LIN {X 0,Y 474.62,Z 424.367,A -85,B 0,C 180,E1 -7430.451,E2 -7430.451} C_VEL
LIN {X 0,Y 474.556,Z 424.367,A -85,B 0,C 180,E1 -7433.225,E2 -7433.225} C_VEL
LIN {X 0,Y 473.902,Z 424.453,A -85,B 0,C 180,E1 -7433.934,E2 -7433.934} C_VEL
LIN {X 0,Y 471.059,Z 424.804,A -85,B 0,C 180,E1 -7435.086,E2 -7435.086} C_VEL
LIN {X 0,Y 468.658,Z 425.105,A -85,B 0,C 180,E1 -7436.015,E2 -7436.015} C_VEL
LIN {X 0,Y 467.644,Z 425.233,A -85,B 0,C 180,E1 -7436.732,E2 -7436.732} C_VEL
LIN {X 0,Y 467.57,Z 425.237,A -85,B 0,C 180,E1 -7436.975,E2 -7436.975} C_VEL
LIN {X 0,Y 467.568,Z 425.238,A -85,B 0,C 180,E1 -7439.266,E2 -7439.266} C_VEL
LIN {X 0,Y 467.577,Z 425.245,A -85,B 0,C 180,E1 -7442.475,E2 -7442.475} C_VEL
LIN {X 0,Y 467.57,Z 425.238,A -85,B 0,C 180,E1 -7445.11,E2 -7445.11} C_VEL
LIN {X 0,Y 467.536,Z 425.244,A -85,B 0,C 180,E1 -7447.926,E2 -7447.926} C_VEL
LIN {X 0,Y 467.622,Z 425.236,A -85,B 0,C 180,E1 -7450.692,E2 -7450.692} C_VEL
LIN {X 0,Y 467.639,Z 425.235,A -85,B 0,C 180,E1 -7454.305,E2 -7454.305} C_VEL
LIN {X 0,Y 467.658,Z 425.228,A -85,B 0,C 180,E1 -7457.854,E2 -7457.854} C_VEL
LIN {X 0,Y 467.669,Z 425.225,A -85,B 0,C 180,E1 -7461.357,E2 -7461.357} C_VEL
LIN {X 0,Y 467.714,Z 425.222,A -85,B 0,C 180,E1 -7463.962,E2 -7463.962} C_VEL
LIN {X 0,Y 467.852,Z 425.202,A -85,B 0,C 180,E1 -7467.417,E2 -7467.417} C_VEL
LIN {X 0,Y 467.88,Z 425.201,A -85,B 0,C 180,E1 -7470,E2 -7470} C_VEL
LIN {X 0,Y 467.848,Z 425.21,A -85,B 0,C 180,E1 -7472.583,E2 -7472.583} C_VEL
LIN {X 0,Y 467.741,Z 425.219,A -85,B 0,C 180,E1 -7476.037,E2 -7476.037} C_VEL
LIN {X 0,Y 467.669,Z 425.232,A -85,B 0,C 180,E1 -7478.643,E2 -7478.643} C_VEL
LIN {X 0,Y 467.657,Z 425.23,A -85,B 0,C 180,E1 -7482.145,E2 -7482.145} C_VEL
LIN {X 0,Y 467.64,Z 425.229,A -85,B 0,C 180,E1 -7485.695,E2 -7485.695} C_VEL
LIN {X 0,Y 467.623,Z 425.231,A -85,B 0,C 180,E1 -7489.307,E2 -7489.307} C_VEL
LIN {X 0,Y 467.535,Z 425.244,A -85,B 0,C 180,E1 -7492.074,E2 -7492.074} C_VEL
LIN {X 0,Y 467.583,Z 425.24,A -85,B 0,C 180,E1 -7494.888,E2 -7494.888} C_VEL
LIN {X 0,Y 467.58,Z 425.237,A -85,B 0,C 180,E1 -7497.771,E2 -7497.771} C_VEL
LIN {X 0,Y 467.568,Z 425.24,A -85,B 0,C 180,E1 -7501.045,E2 -7501.045} C_VEL
LIN {X 0,Y 467.588,Z 425.239,A -85,B 0,C 180,E1 -7504.242,E2 -7504.242} C_VEL
LIN {X 0,Y 467.543,Z 425.242,A -85,B 0,C 180,E1 -7507.185,E2 -7507.185} C_VEL
LIN {X 0,Y 467.569,Z 425.242,A -85,B 0,C 180,E1 -7510.265,E2 -7510.265} C_VEL
LIN {X 0,Y 467.559,Z 425.248,A -85,B 0,C 180,E1 -7512.563,E2 -7512.563} C_VEL
LIN {X 0,Y 467.564,Z 425.241,A -85,B 0,C 180,E1 -7515.052,E2 -7515.052} C_VEL
LIN {X 0,Y 467.572,Z 425.246,A -85,B 0,C 180,E1 -7518.597,E2 -7518.597} C_VEL
LIN {X 0,Y 467.558,Z 425.239,A -85,B 0,C 180,E1 -7521.409,E2 -7521.409} C_VEL
LIN {X 0,Y 467.557,Z 425.243,A -85,B 0,C 180,E1 -7524.261,E2 -7524.261} C_VEL
LIN {X 0,Y 467.581,Z 425.237,A -85,B 0,C 180,E1 -7527.321,E2 -7527.321} C_VEL
LIN {X 0,Y 467.568,Z 425.245,A -85,B 0,C 180,E1 -7530.668,E2 -7530.668} C_VEL
LIN {X 0,Y 467.587,Z 425.237,A -85,B 0,C 180,E1 -7533.198,E2 -7533.198} C_VEL
LIN {X 0,Y 467.59,Z 425.242,A -85,B 0,C 180,E1 -7536.469,E2 -7536.469} C_VEL
LIN {X 0,Y 467.622,Z 425.231,A -85,B 0,C 180,E1 -7539.777,E2 -7539.777} C_VEL
LIN {X 0,Y 467.597,Z 425.241,A -85,B 0,C 180,E1 -7542.506,E2 -7542.506} C_VEL
LIN {X 0,Y 467.604,Z 425.235,A -85,B 0,C 180,E1 -7545.196,E2 -7545.196} C_VEL
LIN {X 0,Y 467.656,Z 425.227,A -85,B 0,C 180,E1 -7547.855,E2 -7547.855} C_VEL
LIN {X 0,Y 467.68,Z 425.224,A -85,B 0,C 180,E1 -7551.357,E2 -7551.357} C_VEL
LIN {X 0,Y 467.723,Z 425.219,A -85,B 0,C 180,E1 -7553.962,E2 -7553.962} C_VEL
LIN {X 0,Y 467.858,Z 425.202,A -85,B 0,C 180,E1 -7557.417,E2 -7557.417} C_VEL
LIN {X 0,Y 467.882,Z 425.2,A -85,B 0,C 180,E1 -7560,E2 -7560} C_VEL
LIN {X 0,Y 467.858,Z 425.209,A -85,B 0,C 180,E1 -7562.583,E2 -7562.583} C_VEL
LIN {X 0,Y 467.742,Z 425.217,A -85,B 0,C 180,E1 -7566.037,E2 -7566.037} C_VEL
LIN {X 0,Y 467.68,Z 425.232,A -85,B 0,C 180,E1 -7568.643,E2 -7568.643} C_VEL
LIN {X 0,Y 467.656,Z 425.229,A -85,B 0,C 180,E1 -7572.146,E2 -7572.146} C_VEL
LIN {X 0,Y 467.639,Z 425.229,A -85,B 0,C 180,E1 -7575.695,E2 -7575.695} C_VEL
LIN {X 0,Y 467.613,Z 425.24,A -85,B 0,C 180,E1 -7578.763,E2 -7578.763} C_VEL
LIN {X 0,Y 467.58,Z 425.238,A -85,B 0,C 180,E1 -7581.268,E2 -7581.268} C_VEL
LIN {X 0,Y 467.568,Z 425.238,A -85,B 0,C 180,E1 -7583.944,E2 -7583.944} C_VEL
LIN {X 0,Y 467.59,Z 425.242,A -85,B 0,C 180,E1 -7586.802,E2 -7586.802} C_VEL
LIN {X 0,Y 467.553,Z 425.24,A -85,B 0,C 180,E1 -7589.738,E2 -7589.738} C_VEL
LIN {X 0,Y 467.583,Z 425.244,A -85,B 0,C 180,E1 -7592.759,E2 -7592.759} C_VEL
LIN {X 0,Y 467.553,Z 425.24,A -85,B 0,C 180,E1 -7595.89,E2 -7595.89} C_VEL
LIN {X 0,Y 467.576,Z 425.24,A -85,B 0,C 180,E1 -7599.146,E2 -7599.146} C_VEL
LIN {X 0,Y 467.587,Z 425.242,A -85,B 0,C 180,E1 -7602.567,E2 -7602.567} C_VEL
LIN {X 0,Y 467.571,Z 425.241,A -85,B 0,C 180,E1 -7605.053,E2 -7605.053} C_VEL
LIN {X 0,Y 467.589,Z 425.236,A -85,B 0,C 180,E1 -7607.44,E2 -7607.44} C_VEL
LIN {X 0,Y 467.582,Z 425.243,A -85,B 0,C 180,E1 -7610.856,E2 -7610.856} C_VEL
LIN {X 0,Y 467.558,Z 425.241,A -85,B 0,C 180,E1 -7614.262,E2 -7614.262} C_VEL
LIN {X 0,Y 467.583,Z 425.238,A -85,B 0,C 180,E1 -7617.321,E2 -7617.321} C_VEL
LIN {X 0,Y 467.57,Z 425.244,A -85,B 0,C 180,E1 -7620.668,E2 -7620.668} C_VEL
LIN {X 0,Y 467.64,Z 425.277,A -85,B 0,C 180,E1 -7621.958,E2 -7621.958} C_VEL
LIN {X 0,Y 470.44,Z 438.906,A -85,B 0,C 180,E1 -7624.327,E2 -7624.327} C_VEL
LIN {X 0,Y 470.495,Z 444.774,A -85,B 0,C 180,E1 -7625.276,E2 -7625.276} C_VEL
LIN {X 0,Y 469.437,Z 466.708,A -85,B 0,C 180,E1 -7628.726,E2 -7628.726} C_VEL
LIN {X 0,Y 468.659,Z 486.966,A -85,B 0,C 180,E1 -7631.871,E2 -7631.871} C_VEL
LIN {X 0,Y 468.408,Z 494.383,A -85,B 0,C 180,E1 -7633.004,E2 -7633.004} C_VEL
LIN {X 0,Y 471.057,Z 514.85,A -85,B 0,C 180,E1 -7633.441,E2 -7633.441} C_VEL
LIN {X 0,Y 470.187,Z 603.81,A -85,B 0,C 180,E1 -7634.92,E2 -7634.92} C_VEL
LIN {X 0,Y 469.824,Z 616.734,A -85,B 0,C 180,E1 -7635.296,E2 -7635.296} C_VEL
LIN {X 0,Y 469.33,Z 629.907,A -85,B 0,C 180,E1 -7635.861,E2 -7635.861} C_VEL
LIN {X 0,Y 468.901,Z 641.86,A -85,B 0,C 180,E1 -7636.567,E2 -7636.567} C_VEL
LIN {X 0,Y 468.404,Z 653.827,A -85,B 0,C 180,E1 -7637.474,E2 -7637.474} C_VEL
LIN {X 0,Y 467.977,Z 663.748,A -85,B 0,C 180,E1 -7638.413,E2 -7638.413} C_VEL
LIN {X 0,Y 467.505,Z 673.902,A -85,B 0,C 180,E1 -7639.607,E2 -7639.607} C_VEL
LIN {X 0,Y 467.18,Z 682.846,A -85,B 0,C 180,E1 -7640.912,E2 -7640.912} C_VEL
LIN {X 0,Y 466.959,Z 689.988,A -85,B 0,C 180,E1 -7642.215,E2 -7642.215} C_VEL
LIN {X 0,Y 466.803,Z 695.821,A -85,B 0,C 180,E1 -7643.552,E2 -7643.552} C_VEL
LIN {X 0,Y 466.779,Z 700.165,A -85,B 0,C 180,E1 -7644.817,E2 -7644.817} C_VEL
LIN {X 0,Y 466.701,Z 702.517,A -85,B 0,C 180,E1 -7645.682,E2 -7645.682} C_VEL
LIN {X 0,Y 466.758,Z 704.438,A -85,B 0,C 180,E1 -7646.547,E2 -7646.547} C_VEL
LIN {X 0,Y 466.775,Z 705.879,A -85,B 0,C 180,E1 -7647.411,E2 -7647.411} C_VEL
LIN {X 0,Y 466.698,Z 706.884,A -85,B 0,C 180,E1 -7648.274,E2 -7648.274} C_VEL
LIN {X 0,Y 466.633,Z 707.487,A -85,B 0,C 180,E1 -7649.137,E2 -7649.137} C_VEL
LIN {X 0,Y 466.624,Z 707.689,A -85,B 0,C 180,E1 -7650,E2 -7650} C_VEL
LIN {X 0,Y 466.634,Z 707.441,A -85,B 0,C 180,E1 -7650.863,E2 -7650.863} C_VEL
LIN {X 0,Y 466.699,Z 706.788,A -85,B 0,C 180,E1 -7651.726,E2 -7651.726} C_VEL
LIN {X 0,Y 466.792,Z 705.732,A -85,B 0,C 180,E1 -7652.589,E2 -7652.589} C_VEL
LIN {X 0,Y 466.772,Z 704.246,A -85,B 0,C 180,E1 -7653.453,E2 -7653.453} C_VEL
LIN {X 0,Y 466.712,Z 701.144,A -85,B 0,C 180,E1 -7654.751,E2 -7654.751} C_VEL
LIN {X 0,Y 466.783,Z 696.966,A -85,B 0,C 180,E1 -7656.05,E2 -7656.05} C_VEL
LIN {X 0,Y 466.939,Z 691.594,A -85,B 0,C 180,E1 -7657.351,E2 -7657.351} C_VEL
LIN {X 0,Y 467.099,Z 684.831,A -85,B 0,C 180,E1 -7658.654,E2 -7658.654} C_VEL
LIN {X 0,Y 467.348,Z 676.43,A -85,B 0,C 180,E1 -7659.959,E2 -7659.959} C_VEL
LIN {X 0,Y 467.714,Z 667.861,A -85,B 0,C 180,E1 -7661.046,E2 -7661.046} C_VEL
LIN {X 0,Y 468.107,Z 658.514,A -85,B 0,C 180,E1 -7662.024,E2 -7662.024} C_VEL
LIN {X 0,Y 468.56,Z 646.916,A -85,B 0,C 180,E1 -7663.002,E2 -7663.002} C_VEL
LIN {X 0,Y 469.023,Z 635.597,A -85,B 0,C 180,E1 -7663.762,E2 -7663.762} C_VEL
LIN {X 0,Y 469.521,Z 623.009,A -85,B 0,C 180,E1 -7664.41,E2 -7664.41} C_VEL
LIN {X 0,Y 469.953,Z 609.708,A -85,B 0,C 180,E1 -7664.894,E2 -7664.894} C_VEL
LIN {X 0,Y 470.286,Z 597.064,A -85,B 0,C 180,E1 -7665.188,E2 -7665.188} C_VEL
LIN {X 0,Y 471.024,Z 514.08,A -85,B 0,C 180,E1 -7666.577,E2 -7666.577} C_VEL
LIN {X 0,Y 468.283,Z 492.11,A -85,B 0,C 180,E1 -7667.095,E2 -7667.095} C_VEL
LIN {X 0,Y 469.001,Z 470.807,A -85,B 0,C 180,E1 -7670.39,E2 -7670.39} C_VEL
LIN {X 0,Y 469.616,Z 456.296,A -85,B 0,C 180,E1 -7672.666,E2 -7672.666} C_VEL
LIN {X 0,Y 470.349,Z 440.454,A -85,B 0,C 180,E1 -7675.205,E2 -7675.205} C_VEL
LIN {X 0,Y 469.688,Z 435.05,A -85,B 0,C 180,E1 -7676.131,E2 -7676.131} C_VEL
LIN {X 0,Y 467.625,Z 425.238,A -85,B 0,C 180,E1 -7677.952,E2 -7677.952} C_VEL
LIN {X 0,Y 467.572,Z 425.248,A -85,B 0,C 180,E1 -7681.045,E2 -7681.045} C_VEL
LIN {X 0,Y 467.592,Z 425.243,A -85,B 0,C 180,E1 -7684.242,E2 -7684.242} C_VEL
LIN {X 0,Y 467.552,Z 425.247,A -85,B 0,C 180,E1 -7687.186,E2 -7687.186} C_VEL
LIN {X 0,Y 467.581,Z 425.241,A -85,B 0,C 180,E1 -7690.265,E2 -7690.265} C_VEL
LIN {X 0,Y 467.59,Z 425.241,A -85,B 0,C 180,E1 -7692.567,E2 -7692.567} C_VEL
LIN {X 0,Y 467.569,Z 425.242,A -85,B 0,C 180,E1 -7695.053,E2 -7695.053} C_VEL
LIN {X 0,Y 467.577,Z 425.245,A -85,B 0,C 180,E1 -7698.597,E2 -7698.597} C_VEL
LIN {X 0,Y 467.562,Z 425.24,A -85,B 0,C 180,E1 -7701.41,E2 -7701.41} C_VEL
LIN {X 0,Y 467.561,Z 425.244,A -85,B 0,C 180,E1 -7704.262,E2 -7704.262} C_VEL
LIN {X 0,Y 467.585,Z 425.236,A -85,B 0,C 180,E1 -7707.321,E2 -7707.321} C_VEL
LIN {X 0,Y 467.554,Z 425.245,A -85,B 0,C 180,E1 -7710.672,E2 -7710.672} C_VEL
LIN {X 0,Y 467.538,Z 425.244,A -85,B 0,C 180,E1 -7713.195,E2 -7713.195} C_VEL
LIN {X 0,Y 467.559,Z 425.245,A -85,B 0,C 180,E1 -7716.056,E2 -7716.056} C_VEL
LIN {X 0,Y 467.551,Z 425.243,A -85,B 0,C 180,E1 -7718.853,E2 -7718.853} C_VEL
LIN {X 0,Y 467.595,Z 425.238,A -85,B 0,C 180,E1 -7721.601,E2 -7721.601} C_VEL
LIN {X 0,Y 467.58,Z 425.243,A -85,B 0,C 180,E1 -7724.303,E2 -7724.303} C_VEL
LIN {X 0,Y 467.644,Z 425.237,A -85,B 0,C 180,E1 -7727.854,E2 -7727.854} C_VEL
LIN {X 0,Y 467.632,Z 425.236,A -85,B 0,C 180,E1 -7731.356,E2 -7731.356} C_VEL
LIN {X 0,Y 467.696,Z 425.231,A -85,B 0,C 180,E1 -7733.962,E2 -7733.962} C_VEL
LIN {X 0,Y 467.669,Z 425.384,A -85,B 0,C 180,E1 -7736.877,E2 -7736.877} C_VEL
LIN {X 0,Y 468.59,Z 429.689,A -85,B 0,C 180,E1 -7738.039,E2 -7738.039} C_VEL
LIN {X 0,Y 471.558,Z 440.896,A -85,B 0,C 180,E1 -7738.372,E2 -7738.372} C_VEL
LIN {X 0,Y 470.383,Z 535.807,A -85,B 0,C 180,E1 -7740,E2 -7740} C_VEL
LIN {X 0,Y 470.125,Z 549.678,A -85,B 0,C 180,E1 -7740.428,E2 -7740.428} C_VEL
LIN {X 0,Y 469.901,Z 561.461,A -85,B 0,C 180,E1 -7740.964,E2 -7740.964} C_VEL
LIN {X 0,Y 469.503,Z 573.791,A -85,B 0,C 180,E1 -7741.716,E2 -7741.716} C_VEL
LIN {X 0,Y 468.962,Z 584.879,A -85,B 0,C 180,E1 -7742.577,E2 -7742.577} C_VEL
LIN {X 0,Y 468.572,Z 593.83,A -85,B 0,C 180,E1 -7743.439,E2 -7743.439} C_VEL
LIN {X 0,Y 468.172,Z 603.023,A -85,B 0,C 180,E1 -7744.52,E2 -7744.52} C_VEL
LIN {X 0,Y 467.851,Z 610.583,A -85,B 0,C 180,E1 -7745.603,E2 -7745.603} C_VEL
LIN {X 0,Y 467.55,Z 617.992,A -85,B 0,C 180,E1 -7746.907,E2 -7746.907} C_VEL
LIN {X 0,Y 467.272,Z 623.956,A -85,B 0,C 180,E1 -7748.215,E2 -7748.215} C_VEL
LIN {X 0,Y 467.067,Z 628.662,A -85,B 0,C 180,E1 -7749.527,E2 -7749.527} C_VEL
LIN {X 0,Y 466.951,Z 632.231,A -85,B 0,C 180,E1 -7750.844,E2 -7750.844} C_VEL
LIN {X 0,Y 466.833,Z 634.764,A -85,B 0,C 180,E1 -7752.167,E2 -7752.167} C_VEL
LIN {X 0,Y 466.732,Z 635.921,A -85,B 0,C 180,E1 -7753.054,E2 -7753.054} C_VEL
LIN {X 0,Y 466.701,Z 636.61,A -85,B 0,C 180,E1 -7753.942,E2 -7753.942} C_VEL
LIN {X 0,Y 466.716,Z 636.823,A -85,B 0,C 180,E1 -7755.475,E2 -7755.475} C_VEL
LIN {X 0,Y 466.695,Z 636.156,A -85,B 0,C 180,E1 -7756.626,E2 -7756.626} C_VEL
LIN {X 0,Y 466.725,Z 635.119,A -85,B 0,C 180,E1 -7757.527,E2 -7757.527} C_VEL
LIN {X 0,Y 466.83,Z 633.563,A -85,B 0,C 180,E1 -7758.476,E2 -7758.476} C_VEL
LIN {X 0,Y 466.92,Z 630.508,A -85,B 0,C 180,E1 -7759.796,E2 -7759.796} C_VEL
LIN {X 0,Y 467.078,Z 626.161,A -85,B 0,C 180,E1 -7761.169,E2 -7761.169} C_VEL
LIN {X 0,Y 467.305,Z 620.456,A -85,B 0,C 180,E1 -7762.551,E2 -7762.551} C_VEL
LIN {X 0,Y 467.609,Z 613.177,A -85,B 0,C 180,E1 -7763.941,E2 -7763.941} C_VEL
LIN {X 0,Y 467.967,Z 605.626,A -85,B 0,C 180,E1 -7765.104,E2 -7765.104} C_VEL
LIN {X 0,Y 468.37,Z 596.274,A -85,B 0,C 180,E1 -7766.273,E2 -7766.273} C_VEL
LIN {X 0,Y 468.81,Z 585.82,A -85,B 0,C 180,E1 -7767.329,E2 -7767.329} C_VEL
LIN {X 0,Y 469.261,Z 575.69,A -85,B 0,C 180,E1 -7768.155,E2 -7768.155} C_VEL
LIN {X 0,Y 469.663,Z 563.942,A -85,B 0,C 180,E1 -7768.916,E2 -7768.916} C_VEL
LIN {X 0,Y 470.051,Z 550.522,A -85,B 0,C 180,E1 -7769.564,E2 -7769.564} C_VEL
LIN {X 0,Y 470.317,Z 538.201,A -85,B 0,C 180,E1 -7769.982,E2 -7769.982} C_VEL
LIN {X 0,Y 470.461,Z 522.713,A -85,B 0,C 180,E1 -7770.292,E2 -7770.292} C_VEL
LIN {X 0,Y 471.2,Z 439.643,A -85,B 0,C 180,E1 -7771.663,E2 -7771.663} C_VEL
LIN {X 0,Y 468.607,Z 429.284,A -85,B 0,C 180,E1 -7771.935,E2 -7771.935} C_VEL
LIN {X 0,Y 467.973,Z 427.129,A -85,B 0,C 180,E1 -7772.018,E2 -7772.018} C_VEL
LIN {X 0,Y 467.621,Z 425.239,A -85,B 0,C 180,E1 -7772.538,E2 -7772.538} C_VEL
LIN {X 0,Y 467.55,Z 425.244,A -85,B 0,C 180,E1 -7775.89,E2 -7775.89} C_VEL
LIN {X 0,Y 467.546,Z 425.241,A -85,B 0,C 180,E1 -7779.148,E2 -7779.148} C_VEL
LIN {X 0,Y 467.567,Z 425.238,A -85,B 0,C 180,E1 -7781.404,E2 -7781.404} C_VEL
LIN {X 0,Y 467.568,Z 425.239,A -85,B 0,C 180,E1 -7785.052,E2 -7785.052} C_VEL
LIN {X 0,Y 467.564,Z 425.242,A -85,B 0,C 180,E1 -7788.725,E2 -7788.725} C_VEL
LIN {X 0,Y 467.543,Z 425.243,A -85,B 0,C 180,E1 -7791.953,E2 -7791.953} C_VEL
LIN {X 0,Y 467.56,Z 425.239,A -85,B 0,C 180,E1 -7795.166,E2 -7795.166} C_VEL
LIN {X 0,Y 467.57,Z 425.237,A -85,B 0,C 180,E1 -7796.975,E2 -7796.975} C_VEL
LIN {X 0,Y 466.933,Z 425.318,A -85,B 0,C 180,E1 -7797.693,E2 -7797.693} C_VEL
LIN {X 0,Y 464.106,Z 425.677,A -85,B 0,C 180,E1 -7798.86,E2 -7798.86} C_VEL
LIN {X 0,Y 461.684,Z 425.981,A -85,B 0,C 180,E1 -7799.8,E2 -7799.8} C_VEL
LIN {X 0,Y 460.62,Z 426.11,A -85,B 0,C 180,E1 -7800.527,E2 -7800.527} C_VEL
LIN {X 0,Y 460.522,Z 426.119,A -85,B 0,C 180,E1 -7800.773,E2 -7800.773} C_VEL
LIN {X 0,Y 460.521,Z 426.116,A -85,B 0,C 180,E1 -7803.732,E2 -7803.732} C_VEL
LIN {X 0,Y 460.546,Z 426.118,A -85,B 0,C 180,E1 -7806.624,E2 -7806.624} C_VEL
LIN {X 0,Y 460.552,Z 426.112,A -85,B 0,C 180,E1 -7809.452,E2 -7809.452} C_VEL
LIN {X 0,Y 460.543,Z 426.118,A -85,B 0,C 180,E1 -7812.229,E2 -7812.229} C_VEL
LIN {X 0,Y 460.562,Z 426.113,A -85,B 0,C 180,E1 -7814.964,E2 -7814.964} C_VEL
LIN {X 0,Y 460.611,Z 426.112,A -85,B 0,C 180,E1 -7818.559,E2 -7818.559} C_VEL
LIN {X 0,Y 460.619,Z 426.104,A -85,B 0,C 180,E1 -7821.223,E2 -7821.223} C_VEL
LIN {X 0,Y 460.679,Z 426.097,A -85,B 0,C 180,E1 -7823.869,E2 -7823.869} C_VEL
LIN {X 0,Y 460.792,Z 426.082,A -85,B 0,C 180,E1 -7827.377,E2 -7827.377} C_VEL
LIN {X 0,Y 460.85,Z 426.077,A -85,B 0,C 180,E1 -7830,E2 -7830} C_VEL
LIN {X 0,Y 460.789,Z 426.089,A -85,B 0,C 180,E1 -7832.622,E2 -7832.622} C_VEL
LIN {X 0,Y 460.706,Z 426.096,A -85,B 0,C 180,E1 -7836.13,E2 -7836.13} C_VEL
LIN {X 0,Y 460.619,Z 426.108,A -85,B 0,C 180,E1 -7838.776,E2 -7838.776} C_VEL
LIN {X 0,Y 460.615,Z 426.112,A -85,B 0,C 180,E1 -7842.445,E2 -7842.445} C_VEL
LIN {X 0,Y 460.601,Z 426.108,A -85,B 0,C 180,E1 -7845.997,E2 -7845.997} C_VEL
LIN {X 0,Y 460.569,Z 426.11,A -85,B 0,C 180,E1 -7849.615,E2 -7849.615} C_VEL
LIN {X 0,Y 460.511,Z 426.124,A -85,B 0,C 180,E1 -7852.428,E2 -7852.428} C_VEL
LIN {X 0,Y 460.549,Z 426.113,A -85,B 0,C 180,E1 -7855.797,E2 -7855.797} C_VEL
LIN {X 0,Y 460.527,Z 426.119,A -85,B 0,C 180,E1 -7858.234,E2 -7858.234} C_VEL
LIN {X 0,Y 460.521,Z 426.116,A -85,B 0,C 180,E1 -7861.283,E2 -7861.283} C_VEL
LIN {X 0,Y 460.531,Z 426.122,A -85,B 0,C 180,E1 -7864.505,E2 -7864.505} C_VEL
LIN {X 0,Y 460.498,Z 426.118,A -85,B 0,C 180,E1 -7867.623,E2 -7867.623} C_VEL
LIN {X 0,Y 460.526,Z 426.118,A -85,B 0,C 180,E1 -7871.011,E2 -7871.011} C_VEL
LIN {X 0,Y 460.511,Z 426.125,A -85,B 0,C 180,E1 -7874.589,E2 -7874.589} C_VEL
LIN {X 0,Y 460.503,Z 426.118,A -85,B 0,C 180,E1 -7877.816,E2 -7877.816} C_VEL
LIN {X 0,Y 460.522,Z 426.118,A -85,B 0,C 180,E1 -7880.136,E2 -7880.136} C_VEL
LIN {X 0,Y 460.472,Z 426.122,A -85,B 0,C 180,E1 -7883.47,E2 -7883.47} C_VEL
LIN {X 0,Y 460.528,Z 426.122,A -85,B 0,C 180,E1 -7886.675,E2 -7886.675} C_VEL
LIN {X 0,Y 460.51,Z 426.117,A -85,B 0,C 180,E1 -7889.76,E2 -7889.76} C_VEL
LIN {X 0,Y 460.558,Z 426.117,A -85,B 0,C 180,E1 -7892.755,E2 -7892.755} C_VEL
LIN {X 0,Y 460.528,Z 426.115,A -85,B 0,C 180,E1 -7895.667,E2 -7895.667} C_VEL
LIN {X 0,Y 460.521,Z 426.124,A -85,B 0,C 180,E1 -7898.578,E2 -7898.578} C_VEL
LIN {X 0,Y 460.585,Z 426.108,A -85,B 0,C 180,E1 -7901.311,E2 -7901.311} C_VEL
LIN {X 0,Y 460.604,Z 426.107,A -85,B 0,C 180,E1 -7904.059,E2 -7904.059} C_VEL
LIN {X 0,Y 460.609,Z 426.105,A -85,B 0,C 180,E1 -7907.666,E2 -7907.666} C_VEL
LIN {X 0,Y 460.627,Z 426.104,A -85,B 0,C 180,E1 -7911.224,E2 -7911.224} C_VEL
LIN {X 0,Y 460.687,Z 426.095,A -85,B 0,C 180,E1 -7913.87,E2 -7913.87} C_VEL
LIN {X 0,Y 460.799,Z 426.082,A -85,B 0,C 180,E1 -7917.378,E2 -7917.378} C_VEL
LIN {X 0,Y 460.852,Z 426.075,A -85,B 0,C 180,E1 -7920,E2 -7920} C_VEL
LIN {X 0,Y 460.823,Z 426.086,A -85,B 0,C 180,E1 -7922.622,E2 -7922.622} C_VEL
LIN {X 0,Y 460.709,Z 426.094,A -85,B 0,C 180,E1 -7926.13,E2 -7926.13} C_VEL
LIN {X 0,Y 460.627,Z 426.109,A -85,B 0,C 180,E1 -7928.776,E2 -7928.776} C_VEL
LIN {X 0,Y 460.613,Z 426.109,A -85,B 0,C 180,E1 -7932.445,E2 -7932.445} C_VEL
LIN {X 0,Y 460.6,Z 426.107,A -85,B 0,C 180,E1 -7935.998,E2 -7935.998} C_VEL
LIN {X 0,Y 460.568,Z 426.11,A -85,B 0,C 180,E1 -7939.616,E2 -7939.616} C_VEL
LIN {X 0,Y 460.511,Z 426.122,A -85,B 0,C 180,E1 -7942.429,E2 -7942.429} C_VEL
LIN {X 0,Y 460.548,Z 426.112,A -85,B 0,C 180,E1 -7945.797,E2 -7945.797} C_VEL
LIN {X 0,Y 460.549,Z 426.115,A -85,B 0,C 180,E1 -7948.233,E2 -7948.233} C_VEL
LIN {X 0,Y 460.521,Z 426.117,A -85,B 0,C 180,E1 -7951.283,E2 -7951.283} C_VEL
LIN {X 0,Y 460.532,Z 426.12,A -85,B 0,C 180,E1 -7954.506,E2 -7954.506} C_VEL
LIN {X 0,Y 460.501,Z 426.118,A -85,B 0,C 180,E1 -7957.623,E2 -7957.623} C_VEL
LIN {X 0,Y 460.539,Z 426.116,A -85,B 0,C 180,E1 -7960.269,E2 -7960.269} C_VEL
LIN {X 0,Y 460.5,Z 426.119,A -85,B 0,C 180,E1 -7963.376,E2 -7963.376} C_VEL
LIN {X 0,Y 460.509,Z 426.124,A -85,B 0,C 180,E1 -7966.626,E2 -7966.626} C_VEL
LIN {X 0,Y 460.542,Z 426.113,A -85,B 0,C 180,E1 -7969.731,E2 -7969.731} C_VEL
LIN {X 0,Y 460.497,Z 426.124,A -85,B 0,C 180,E1 -7972.525,E2 -7972.525} C_VEL
LIN {X 0,Y 460.546,Z 426.113,A -85,B 0,C 180,E1 -7975.624,E2 -7975.624} C_VEL
LIN {X 0,Y 460.538,Z 426.12,A -85,B 0,C 180,E1 -7978.745,E2 -7978.745} C_VEL
LIN {X 0,Y 460.605,Z 426.187,A -85,B 0,C 180,E1 -7981.74,E2 -7981.74} C_VEL
LIN {X 0,Y 463.416,Z 439.815,A -85,B 0,C 180,E1 -7984.151,E2 -7984.151} C_VEL
LIN {X 0,Y 463.601,Z 444.235,A -85,B 0,C 180,E1 -7984.883,E2 -7984.883} C_VEL
LIN {X 0,Y 462.569,Z 465.271,A -85,B 0,C 180,E1 -7988.248,E2 -7988.248} C_VEL
LIN {X 0,Y 461.743,Z 484.989,A -85,B 0,C 180,E1 -7991.36,E2 -7991.36} C_VEL
LIN {X 0,Y 461.405,Z 493.829,A -85,B 0,C 180,E1 -7992.745,E2 -7992.745} C_VEL
LIN {X 0,Y 464.205,Z 515.194,A -85,B 0,C 180,E1 -7993.22,E2 -7993.22} C_VEL
LIN {X 0,Y 463.288,Z 603.461,A -85,B 0,C 180,E1 -7994.718,E2 -7994.718} C_VEL
LIN {X 0,Y 462.91,Z 616.315,A -85,B 0,C 180,E1 -7995.099,E2 -7995.099} C_VEL
LIN {X 0,Y 462.38,Z 628.897,A -85,B 0,C 180,E1 -7995.644,E2 -7995.644} C_VEL
LIN {X 0,Y 461.936,Z 640.989,A -85,B 0,C 180,E1 -7996.36,E2 -7996.36} C_VEL
LIN {X 0,Y 461.397,Z 652.905,A -85,B 0,C 180,E1 -7997.27,E2 -7997.27} C_VEL
LIN {X 0,Y 460.92,Z 663.01,A -85,B 0,C 180,E1 -7998.233,E2 -7998.233} C_VEL
LIN {X 0,Y 460.564,Z 671.563,A -85,B 0,C 180,E1 -7999.227,E2 -7999.227} C_VEL
LIN {X 0,Y 460.169,Z 680.827,A -85,B 0,C 180,E1 -8000.551,E2 -8000.551} C_VEL
LIN {X 0,Y 459.929,Z 688.29,A -85,B 0,C 180,E1 -8001.875,E2 -8001.875} C_VEL
LIN {X 0,Y 459.777,Z 693.339,A -85,B 0,C 180,E1 -8002.976,E2 -8002.976} C_VEL
LIN {X 0,Y 459.718,Z 698.234,A -85,B 0,C 180,E1 -8004.297,E2 -8004.297} C_VEL
LIN {X 0,Y 459.611,Z 701.964,A -85,B 0,C 180,E1 -8005.615,E2 -8005.615} C_VEL
LIN {X 0,Y 459.688,Z 703.892,A -85,B 0,C 180,E1 -8006.494,E2 -8006.494} C_VEL
LIN {X 0,Y 459.689,Z 705.339,A -85,B 0,C 180,E1 -8007.371,E2 -8007.371} C_VEL
LIN {X 0,Y 459.637,Z 706.347,A -85,B 0,C 180,E1 -8008.248,E2 -8008.248} C_VEL
LIN {X 0,Y 459.566,Z 706.951,A -85,B 0,C 180,E1 -8009.124,E2 -8009.124} C_VEL
LIN {X 0,Y 459.554,Z 707.152,A -85,B 0,C 180,E1 -8010,E2 -8010} C_VEL
LIN {X 0,Y 459.567,Z 706.903,A -85,B 0,C 180,E1 -8010.877,E2 -8010.877} C_VEL
LIN {X 0,Y 459.638,Z 706.246,A -85,B 0,C 180,E1 -8011.753,E2 -8011.753} C_VEL
LIN {X 0,Y 459.705,Z 705.184,A -85,B 0,C 180,E1 -8012.629,E2 -8012.629} C_VEL
LIN {X 0,Y 459.701,Z 703.693,A -85,B 0,C 180,E1 -8013.506,E2 -8013.506} C_VEL
LIN {X 0,Y 459.642,Z 700.582,A -85,B 0,C 180,E1 -8014.824,E2 -8014.824} C_VEL
LIN {X 0,Y 459.719,Z 696.391,A -85,B 0,C 180,E1 -8016.144,E2 -8016.144} C_VEL
LIN {X 0,Y 459.844,Z 690.999,A -85,B 0,C 180,E1 -8017.465,E2 -8017.465} C_VEL
LIN {X 0,Y 460.013,Z 684.213,A -85,B 0,C 180,E1 -8018.788,E2 -8018.788} C_VEL
LIN {X 0,Y 460.307,Z 675.806,A -85,B 0,C 180,E1 -8020.113,E2 -8020.113} C_VEL
LIN {X 0,Y 460.694,Z 667.232,A -85,B 0,C 180,E1 -8021.216,E2 -8021.216} C_VEL
LIN {X 0,Y 461.124,Z 657.884,A -85,B 0,C 180,E1 -8022.209,E2 -8022.209} C_VEL
LIN {X 0,Y 461.592,Z 646.28,A -85,B 0,C 180,E1 -8023.202,E2 -8023.202} C_VEL
LIN {X 0,Y 462.086,Z 634.943,A -85,B 0,C 180,E1 -8023.972,E2 -8023.972} C_VEL
LIN {X 0,Y 462.626,Z 622.335,A -85,B 0,C 180,E1 -8024.629,E2 -8024.629} C_VEL
LIN {X 0,Y 463.089,Z 609.029,A -85,B 0,C 180,E1 -8025.12,E2 -8025.12} C_VEL
LIN {X 0,Y 463.441,Z 596.402,A -85,B 0,C 180,E1 -8025.418,E2 -8025.418} C_VEL
LIN {X 0,Y 464.252,Z 515.176,A -85,B 0,C 180,E1 -8026.81,E2 -8026.81} C_VEL
LIN {X 0,Y 461.299,Z 491.585,A -85,B 0,C 180,E1 -8027.366,E2 -8027.366} C_VEL
LIN {X 0,Y 462.021,Z 471.809,A -85,B 0,C 180,E1 -8030.479,E2 -8030.479} C_VEL
LIN {X 0,Y 462.782,Z 454.498,A -85,B 0,C 180,E1 -8033.257,E2 -8033.257} C_VEL
LIN {X 0,Y 463.461,Z 441.594,A -85,B 0,C 180,E1 -8035.366,E2 -8035.366} C_VEL
LIN {X 0,Y 462.337,Z 434.292,A -85,B 0,C 180,E1 -8036.668,E2 -8036.668} C_VEL
LIN {X 0,Y 460.591,Z 426.114,A -85,B 0,C 180,E1 -8038.231,E2 -8038.231} C_VEL
LIN {X 0,Y 460.525,Z 426.127,A -85,B 0,C 180,E1 -8041.283,E2 -8041.283} C_VEL
LIN {X 0,Y 460.536,Z 426.124,A -85,B 0,C 180,E1 -8044.506,E2 -8044.506} C_VEL
LIN {X 0,Y 460.505,Z 426.122,A -85,B 0,C 180,E1 -8047.623,E2 -8047.623} C_VEL
LIN {X 0,Y 460.545,Z 426.117,A -85,B 0,C 180,E1 -8050.27,E2 -8050.27} C_VEL
LIN {X 0,Y 460.502,Z 426.121,A -85,B 0,C 180,E1 -8053.376,E2 -8053.376} C_VEL
LIN {X 0,Y 460.512,Z 426.125,A -85,B 0,C 180,E1 -8056.626,E2 -8056.626} C_VEL
LIN {X 0,Y 460.54,Z 426.115,A -85,B 0,C 180,E1 -8059.732,E2 -8059.732} C_VEL
LIN {X 0,Y 460.5,Z 426.127,A -85,B 0,C 180,E1 -8062.525,E2 -8062.525} C_VEL
LIN {X 0,Y 460.549,Z 426.112,A -85,B 0,C 180,E1 -8065.624,E2 -8065.624} C_VEL
LIN {X 0,Y 460.541,Z 426.118,A -85,B 0,C 180,E1 -8068.745,E2 -8068.745} C_VEL
LIN {X 0,Y 460.511,Z 426.12,A -85,B 0,C 180,E1 -8071.764,E2 -8071.764} C_VEL
LIN {X 0,Y 460.526,Z 426.12,A -85,B 0,C 180,E1 -8074.703,E2 -8074.703} C_VEL
LIN {X 0,Y 460.509,Z 426.121,A -85,B 0,C 180,E1 -8077.571,E2 -8077.571} C_VEL
LIN {X 0,Y 460.528,Z 426.116,A -85,B 0,C 180,E1 -8081.115,E2 -8081.115} C_VEL
LIN {X 0,Y 460.523,Z 426.123,A -85,B 0,C 180,E1 -8084.056,E2 -8084.056} C_VEL
LIN {X 0,Y 460.605,Z 426.112,A -85,B 0,C 180,E1 -8087.666,E2 -8087.666} C_VEL
LIN {X 0,Y 460.587,Z 426.113,A -85,B 0,C 180,E1 -8091.223,E2 -8091.223} C_VEL
LIN {X 0,Y 460.662,Z 426.107,A -85,B 0,C 180,E1 -8093.869,E2 -8093.869} C_VEL
LIN {X 0,Y 460.559,Z 426.26,A -85,B 0,C 180,E1 -8096.61,E2 -8096.61} C_VEL
LIN {X 0,Y 461.587,Z 430.406,A -85,B 0,C 180,E1 -8097.75,E2 -8097.75} C_VEL
LIN {X 0,Y 464.554,Z 440.707,A -85,B 0,C 180,E1 -8098.07,E2 -8098.07} C_VEL
LIN {X 0,Y 464.81,Z 442.718,A -85,B 0,C 180,E1 -8098.118,E2 -8098.118} C_VEL
LIN {X 0,Y 463.567,Z 535.835,A -85,B 0,C 180,E1 -8099.761,E2 -8099.761} C_VEL
LIN {X 0,Y 463.312,Z 549.695,A -85,B 0,C 180,E1 -8100.19,E2 -8100.19} C_VEL
LIN {X 0,Y 463.042,Z 562.165,A -85,B 0,C 180,E1 -8100.761,E2 -8100.761} C_VEL
LIN {X 0,Y 462.607,Z 574.481,A -85,B 0,C 180,E1 -8101.523,E2 -8101.523} C_VEL
LIN {X 0,Y 462.059,Z 585.548,A -85,B 0,C 180,E1 -8102.397,E2 -8102.397} C_VEL
LIN {X 0,Y 461.636,Z 594.495,A -85,B 0,C 180,E1 -8103.273,E2 -8103.273} C_VEL
LIN {X 0,Y 461.221,Z 603.671,A -85,B 0,C 180,E1 -8104.369,E2 -8104.369} C_VEL
LIN {X 0,Y 460.809,Z 612.571,A -85,B 0,C 180,E1 -8105.689,E2 -8105.689} C_VEL
LIN {X 0,Y 460.505,Z 619.739,A -85,B 0,C 180,E1 -8107.013,E2 -8107.013} C_VEL
LIN {X 0,Y 460.196,Z 625.463,A -85,B 0,C 180,E1 -8108.342,E2 -8108.342} C_VEL
LIN {X 0,Y 460.013,Z 629.937,A -85,B 0,C 180,E1 -8109.675,E2 -8109.675} C_VEL
LIN {X 0,Y 459.909,Z 632.29,A -85,B 0,C 180,E1 -8110.566,E2 -8110.566} C_VEL
LIN {X 0,Y 459.773,Z 635.058,A -85,B 0,C 180,E1 -8111.958,E2 -8111.958} C_VEL
LIN {X 0,Y 459.639,Z 636.68,A -85,B 0,C 180,E1 -8113.259,E2 -8113.259} C_VEL
LIN {X 0,Y 459.622,Z 637.276,A -85,B 0,C 180,E1 -8114.161,E2 -8114.161} C_VEL
LIN {X 0,Y 459.633,Z 637.34,A -85,B 0,C 180,E1 -8115.569,E2 -8115.569} C_VEL
LIN {X 0,Y 459.618,Z 636.45,A -85,B 0,C 180,E1 -8116.89,E2 -8116.89} C_VEL
LIN {X 0,Y 459.678,Z 635.311,A -85,B 0,C 180,E1 -8117.805,E2 -8117.805} C_VEL
LIN {X 0,Y 459.782,Z 632.692,A -85,B 0,C 180,E1 -8119.186,E2 -8119.186} C_VEL
LIN {X 0,Y 459.959,Z 628.932,A -85,B 0,C 180,E1 -8120.575,E2 -8120.575} C_VEL
LIN {X 0,Y 460.137,Z 623.885,A -85,B 0,C 180,E1 -8121.975,E2 -8121.975} C_VEL
LIN {X 0,Y 460.442,Z 617.385,A -85,B 0,C 180,E1 -8123.382,E2 -8123.382} C_VEL
LIN {X 0,Y 460.765,Z 610.634,A -85,B 0,C 180,E1 -8124.56,E2 -8124.56} C_VEL
LIN {X 0,Y 461.119,Z 602.954,A -85,B 0,C 180,E1 -8125.666,E2 -8125.666} C_VEL
LIN {X 0,Y 461.56,Z 593.225,A -85,B 0,C 180,E1 -8126.814,E2 -8126.814} C_VEL
LIN {X 0,Y 462.057,Z 581.807,A -85,B 0,C 180,E1 -8127.886,E2 -8127.886} C_VEL
LIN {X 0,Y 462.507,Z 570.619,A -85,B 0,C 180,E1 -8128.722,E2 -8128.722} C_VEL
LIN {X 0,Y 462.967,Z 558.101,A -85,B 0,C 180,E1 -8129.437,E2 -8129.437} C_VEL
LIN {X 0,Y 463.257,Z 545.22,A -85,B 0,C 180,E1 -8129.98,E2 -8129.98} C_VEL
LIN {X 0,Y 463.489,Z 531.872,A -85,B 0,C 180,E1 -8130.346,E2 -8130.346} C_VEL
LIN {X 0,Y 464.509,Z 441.27,A -85,B 0,C 180,E1 -8131.878,E2 -8131.878} C_VEL
LIN {X 0,Y 462.044,Z 431.446,A -85,B 0,C 180,E1 -8132.14,E2 -8132.14} C_VEL
LIN {X 0,Y 460.849,Z 427.615,A -85,B 0,C 180,E1 -8132.259,E2 -8132.259} C_VEL
LIN {X 0,Y 460.557,Z 426.119,A -85,B 0,C 180,E1 -8132.669,E2 -8132.669} C_VEL
LIN {X 0,Y 460.507,Z 426.119,A -85,B 0,C 180,E1 -8135.446,E2 -8135.446} C_VEL
LIN {X 0,Y 460.495,Z 426.121,A -85,B 0,C 180,E1 -8138.889,E2 -8138.889} C_VEL
LIN {X 0,Y 460.512,Z 426.117,A -85,B 0,C 180,E1 -8141.599,E2 -8141.599} C_VEL
LIN {X 0,Y 460.514,Z 426.122,A -85,B 0,C 180,E1 -8144.589,E2 -8144.589} C_VEL
LIN {X 0,Y 460.478,Z 426.122,A -85,B 0,C 180,E1 -8147.813,E2 -8147.813} C_VEL
LIN {X 0,Y 460.513,Z 426.121,A -85,B 0,C 180,E1 -8150.135,E2 -8150.135} C_VEL
LIN {X 0,Y 460.463,Z 426.123,A -85,B 0,C 180,E1 -8153.469,E2 -8153.469} C_VEL
LIN {X 0,Y 460.53,Z 426.119,A -85,B 0,C 180,E1 -8156.675,E2 -8156.675} C_VEL
LIN {X 0,Y 460.506,Z 426.118,A -85,B 0,C 180,E1 -8159.759,E2 -8159.759} C_VEL
LIN {X 0,Y 460.522,Z 426.119,A -85,B 0,C 180,E1 -8160.773,E2 -8160.773} C_VEL
LIN {X 0,Y 459.828,Z 426.202,A -85,B 0,C 180,E1 -8161.504,E2 -8161.504} C_VEL
LIN {X 0,Y 456.982,Z 426.561,A -85,B 0,C 180,E1 -8162.69,E2 -8162.69} C_VEL
LIN {X 0,Y 454.591,Z 426.861,A -85,B 0,C 180,E1 -8163.647,E2 -8163.647} C_VEL
LIN {X 0,Y 453.564,Z 426.99,A -85,B 0,C 180,E1 -8164.386,E2 -8164.386} C_VEL
LIN {X 0,Y 453.479,Z 426.995,A -85,B 0,C 180,E1 -8164.636,E2 -8164.636} C_VEL
LIN {X 0,Y 453.48,Z 426.993,A -85,B 0,C 180,E1 -8167.204,E2 -8167.204} C_VEL
LIN {X 0,Y 453.505,Z 426.993,A -85,B 0,C 180,E1 -8170.066,E2 -8170.066} C_VEL
LIN {X 0,Y 453.493,Z 426.994,A -85,B 0,C 180,E1 -8172.875,E2 -8172.875} C_VEL
LIN {X 0,Y 453.509,Z 426.989,A -85,B 0,C 180,E1 -8175.643,E2 -8175.643} C_VEL
LIN {X 0,Y 453.56,Z 426.99,A -85,B 0,C 180,E1 -8178.379,E2 -8178.379} C_VEL
LIN {X 0,Y 453.585,Z 426.981,A -85,B 0,C 180,E1 -8181.086,E2 -8181.086} C_VEL
LIN {X 0,Y 453.645,Z 426.973,A -85,B 0,C 180,E1 -8183.774,E2 -8183.774} C_VEL
LIN {X 0,Y 453.736,Z 426.961,A -85,B 0,C 180,E1 -8187.336,E2 -8187.336} C_VEL
LIN {X 0,Y 453.819,Z 426.953,A -85,B 0,C 180,E1 -8190,E2 -8190} C_VEL
LIN {X 0,Y 453.732,Z 426.967,A -85,B 0,C 180,E1 -8192.663,E2 -8192.663} C_VEL
LIN {X 0,Y 453.673,Z 426.973,A -85,B 0,C 180,E1 -8196.225,E2 -8196.225} C_VEL
LIN {X 0,Y 453.585,Z 426.983,A -85,B 0,C 180,E1 -8198.913,E2 -8198.913} C_VEL
LIN {X 0,Y 453.565,Z 426.99,A -85,B 0,C 180,E1 -8202.529,E2 -8202.529} C_VEL
LIN {X 0,Y 453.545,Z 426.989,A -85,B 0,C 180,E1 -8206.196,E2 -8206.196} C_VEL
LIN {X 0,Y 453.518,Z 426.99,A -85,B 0,C 180,E1 -8209.039,E2 -8209.039} C_VEL
LIN {X 0,Y 453.477,Z 426.994,A -85,B 0,C 180,E1 -8211.836,E2 -8211.836} C_VEL
LIN {X 0,Y 453.5,Z 426.996,A -85,B 0,C 180,E1 -8214.735,E2 -8214.735} C_VEL
LIN {X 0,Y 453.506,Z 426.991,A -85,B 0,C 180,E1 -8217.953,E2 -8217.953} C_VEL
LIN {X 0,Y 453.475,Z 426.999,A -85,B 0,C 180,E1 -8220.759,E2 -8220.759} C_VEL
LIN {X 0,Y 453.476,Z 426.994,A -85,B 0,C 180,E1 -8223.912,E2 -8223.912} C_VEL
LIN {X 0,Y 453.449,Z 426.998,A -85,B 0,C 180,E1 -8227.19,E2 -8227.19} C_VEL
LIN {X 0,Y 453.492,Z 426.999,A -85,B 0,C 180,E1 -8230.609,E2 -8230.609} C_VEL
LIN {X 0,Y 453.459,Z 426.999,A -85,B 0,C 180,E1 -8234.222,E2 -8234.222} C_VEL
LIN {X 0,Y 453.447,Z 427,A -85,B 0,C 180,E1 -8237.003,E2 -8237.003} C_VEL
LIN {X 0,Y 453.493,Z 426.991,A -85,B 0,C 180,E1 -8239.409,E2 -8239.409} C_VEL
LIN {X 0,Y 453.445,Z 427.001,A -85,B 0,C 180,E1 -8242.228,E2 -8242.228} C_VEL
LIN {X 0,Y 453.486,Z 426.993,A -85,B 0,C 180,E1 -8245.223,E2 -8245.223} C_VEL
LIN {X 0,Y 453.466,Z 427.001,A -85,B 0,C 180,E1 -8248.475,E2 -8248.475} C_VEL
LIN {X 0,Y 453.528,Z 426.988,A -85,B 0,C 180,E1 -8252.041,E2 -8252.041} C_VEL
LIN {X 0,Y 453.497,Z 426.992,A -85,B 0,C 180,E1 -8255.265,E2 -8255.265} C_VEL
LIN {X 0,Y 453.48,Z 426.998,A -85,B 0,C 180,E1 -8258.415,E2 -8258.415} C_VEL
LIN {X 0,Y 453.521,Z 426.991,A -85,B 0,C 180,E1 -8261.009,E2 -8261.009} C_VEL
LIN {X 0,Y 453.568,Z 426.982,A -85,B 0,C 180,E1 -8263.88,E2 -8263.88} C_VEL
LIN {X 0,Y 453.563,Z 426.983,A -85,B 0,C 180,E1 -8267.471,E2 -8267.471} C_VEL
LIN {X 0,Y 453.59,Z 426.982,A -85,B 0,C 180,E1 -8271.087,E2 -8271.087} C_VEL
LIN {X 0,Y 453.653,Z 426.971,A -85,B 0,C 180,E1 -8273.774,E2 -8273.774} C_VEL
LIN {X 0,Y 453.743,Z 426.961,A -85,B 0,C 180,E1 -8277.337,E2 -8277.337} C_VEL
LIN {X 0,Y 453.823,Z 426.951,A -85,B 0,C 180,E1 -8280,E2 -8280} C_VEL
LIN {X 0,Y 453.763,Z 426.966,A -85,B 0,C 180,E1 -8282.663,E2 -8282.663} C_VEL
LIN {X 0,Y 453.677,Z 426.971,A -85,B 0,C 180,E1 -8286.225,E2 -8286.225} C_VEL
LIN {X 0,Y 453.59,Z 426.984,A -85,B 0,C 180,E1 -8288.913,E2 -8288.913} C_VEL
LIN {X 0,Y 453.563,Z 426.989,A -85,B 0,C 180,E1 -8292.529,E2 -8292.529} C_VEL
LIN {X 0,Y 453.544,Z 426.987,A -85,B 0,C 180,E1 -8296.196,E2 -8296.196} C_VEL
LIN {X 0,Y 453.517,Z 426.992,A -85,B 0,C 180,E1 -8299.04,E2 -8299.04} C_VEL
LIN {X 0,Y 453.476,Z 426.993,A -85,B 0,C 180,E1 -8301.836,E2 -8301.836} C_VEL
LIN {X 0,Y 453.503,Z 426.998,A -85,B 0,C 180,E1 -8304.735,E2 -8304.735} C_VEL
LIN {X 0,Y 453.528,Z 426.987,A -85,B 0,C 180,E1 -8307.959,E2 -8307.959} C_VEL
LIN {X 0,Y 453.466,Z 426.995,A -85,B 0,C 180,E1 -8311.525,E2 -8311.525} C_VEL
LIN {X 0,Y 453.487,Z 426.999,A -85,B 0,C 180,E1 -8314.778,E2 -8314.778} C_VEL
LIN {X 0,Y 453.463,Z 426.998,A -85,B 0,C 180,E1 -8318.312,E2 -8318.312} C_VEL
LIN {X 0,Y 453.494,Z 426.998,A -85,B 0,C 180,E1 -8320.609,E2 -8320.609} C_VEL
LIN {X 0,Y 453.456,Z 426.998,A -85,B 0,C 180,E1 -8323.244,E2 -8323.244} C_VEL
LIN {X 0,Y 453.472,Z 426.994,A -85,B 0,C 180,E1 -8325.78,E2 -8325.78} C_VEL
LIN {X 0,Y 453.494,Z 426.992,A -85,B 0,C 180,E1 -8329.391,E2 -8329.391} C_VEL
LIN {X 0,Y 453.448,Z 426.999,A -85,B 0,C 180,E1 -8332.228,E2 -8332.228} C_VEL
LIN {X 0,Y 453.487,Z 426.995,A -85,B 0,C 180,E1 -8335.223,E2 -8335.223} C_VEL
LIN {X 0,Y 453.467,Z 426.999,A -85,B 0,C 180,E1 -8338.475,E2 -8338.475} C_VEL
LIN {X 0,Y 453.554,Z 427.119,A -85,B 0,C 180,E1 -8341.526,E2 -8341.526} C_VEL
LIN {X 0,Y 456.4,Z 440.722,A -85,B 0,C 180,E1 -8343.969,E2 -8343.969} C_VEL
LIN {X 0,Y 456.709,Z 445.082,A -85,B 0,C 180,E1 -8344.711,E2 -8344.711} C_VEL
LIN {X 0,Y 455.658,Z 465.291,A -85,B 0,C 180,E1 -8347.993,E2 -8347.993} C_VEL
LIN {X 0,Y 454.71,Z 485.884,A -85,B 0,C 180,E1 -8351.294,E2 -8351.294} C_VEL
LIN {X 0,Y 454.407,Z 493.373,A -85,B 0,C 180,E1 -8352.487,E2 -8352.487} C_VEL
LIN {X 0,Y 457.354,Z 516.056,A -85,B 0,C 180,E1 -8352.997,E2 -8352.997} C_VEL
LIN {X 0,Y 456.39,Z 602.928,A -85,B 0,C 180,E1 -8354.51,E2 -8354.51} C_VEL
LIN {X 0,Y 455.999,Z 615.778,A -85,B 0,C 180,E1 -8354.897,E2 -8354.897} C_VEL
LIN {X 0,Y 455.431,Z 628.919,A -85,B 0,C 180,E1 -8355.478,E2 -8355.478} C_VEL
LIN {X 0,Y 454.979,Z 640.075,A -85,B 0,C 180,E1 -8356.148,E2 -8356.148} C_VEL
LIN {X 0,Y 454.406,Z 652.074,A -85,B 0,C 180,E1 -8357.071,E2 -8357.071} C_VEL
LIN {X 0,Y 453.848,Z 662.239,A -85,B 0,C 180,E1 -8358.047,E2 -8358.047} C_VEL
LIN {X 0,Y 453.534,Z 670.859,A -85,B 0,C 180,E1 -8359.058,E2 -8359.058} C_VEL
LIN {X 0,Y 453.117,Z 680.169,A -85,B 0,C 180,E1 -8360.402,E2 -8360.402} C_VEL
LIN {X 0,Y 452.85,Z 687.66,A -85,B 0,C 180,E1 -8361.747,E2 -8361.747} C_VEL
LIN {X 0,Y 452.719,Z 692.736,A -85,B 0,C 180,E1 -8362.866,E2 -8362.866} C_VEL
LIN {X 0,Y 452.616,Z 697.648,A -85,B 0,C 180,E1 -8364.208,E2 -8364.208} C_VEL
LIN {X 0,Y 452.527,Z 701.397,A -85,B 0,C 180,E1 -8365.547,E2 -8365.547} C_VEL
LIN {X 0,Y 452.601,Z 703.332,A -85,B 0,C 180,E1 -8366.439,E2 -8366.439} C_VEL
LIN {X 0,Y 452.608,Z 704.791,A -85,B 0,C 180,E1 -8367.33,E2 -8367.33} C_VEL
LIN {X 0,Y 452.577,Z 705.805,A -85,B 0,C 180,E1 -8368.221,E2 -8368.221} C_VEL
LIN {X 0,Y 452.501,Z 706.41,A -85,B 0,C 180,E1 -8369.11,E2 -8369.11} C_VEL
LIN {X 0,Y 452.486,Z 706.614,A -85,B 0,C 180,E1 -8370,E2 -8370} C_VEL
LIN {X 0,Y 452.502,Z 706.367,A -85,B 0,C 180,E1 -8370.89,E2 -8370.89} C_VEL
LIN {X 0,Y 452.578,Z 705.706,A -85,B 0,C 180,E1 -8371.78,E2 -8371.78} C_VEL
LIN {X 0,Y 452.623,Z 704.638,A -85,B 0,C 180,E1 -8372.67,E2 -8372.67} C_VEL
LIN {X 0,Y 452.614,Z 703.144,A -85,B 0,C 180,E1 -8373.561,E2 -8373.561} C_VEL
LIN {X 0,Y 452.575,Z 700.027,A -85,B 0,C 180,E1 -8374.9,E2 -8374.9} C_VEL
LIN {X 0,Y 452.629,Z 695.172,A -85,B 0,C 180,E1 -8376.416,E2 -8376.416} C_VEL
LIN {X 0,Y 452.778,Z 689.382,A -85,B 0,C 180,E1 -8377.806,E2 -8377.806} C_VEL
LIN {X 0,Y 453.012,Z 682.367,A -85,B 0,C 180,E1 -8379.15,E2 -8379.15} C_VEL
LIN {X 0,Y 453.338,Z 673.649,A -85,B 0,C 180,E1 -8380.496,E2 -8380.496} C_VEL
LIN {X 0,Y 453.763,Z 663.676,A -85,B 0,C 180,E1 -8381.729,E2 -8381.729} C_VEL
LIN {X 0,Y 454.275,Z 653.246,A -85,B 0,C 180,E1 -8382.776,E2 -8382.776} C_VEL
LIN {X 0,Y 454.781,Z 642.704,A -85,B 0,C 180,E1 -8383.631,E2 -8383.631} C_VEL
LIN {X 0,Y 455.313,Z 630.448,A -85,B 0,C 180,E1 -8384.413,E2 -8384.413} C_VEL
LIN {X 0,Y 455.937,Z 617.773,A -85,B 0,C 180,E1 -8385.02,E2 -8385.02} C_VEL
LIN {X 0,Y 456.365,Z 605.649,A -85,B 0,C 180,E1 -8385.435,E2 -8385.435} C_VEL
LIN {X 0,Y 456.638,Z 589.497,A -85,B 0,C 180,E1 -8385.768,E2 -8385.768} C_VEL
LIN {X 0,Y 457.433,Z 515.156,A -85,B 0,C 180,E1 -8387.082,E2 -8387.082} C_VEL
LIN {X 0,Y 454.344,Z 490.853,A -85,B 0,C 180,E1 -8387.685,E2 -8387.685} C_VEL
LIN {X 0,Y 455.085,Z 471.425,A -85,B 0,C 180,E1 -8390.806,E2 -8390.806} C_VEL
LIN {X 0,Y 455.866,Z 455.606,A -85,B 0,C 180,E1 -8393.39,E2 -8393.39} C_VEL
LIN {X 0,Y 456.579,Z 442.787,A -85,B 0,C 180,E1 -8395.531,E2 -8395.531} C_VEL
LIN {X 0,Y 455.429,Z 435.637,A -85,B 0,C 180,E1 -8396.832,E2 -8396.832} C_VEL
LIN {X 0,Y 453.532,Z 426.993,A -85,B 0,C 180,E1 -8398.515,E2 -8398.515} C_VEL
LIN {X 0,Y 453.468,Z 427.004,A -85,B 0,C 180,E1 -8401.8,E2 -8401.8} C_VEL
LIN {X 0,Y 453.484,Z 427.004,A -85,B 0,C 180,E1 -8404.989,E2 -8404.989} C_VEL
LIN {X 0,Y 453.468,Z 426.999,A -85,B 0,C 180,E1 -8408.312,E2 -8408.312} C_VEL
LIN {X 0,Y 453.498,Z 426.997,A -85,B 0,C 180,E1 -8410.609,E2 -8410.609} C_VEL
LIN {X 0,Y 453.458,Z 427,A -85,B 0,C 180,E1 -8413.244,E2 -8413.244} C_VEL
LIN {X 0,Y 453.464,Z 426.996,A -85,B 0,C 180,E1 -8415.778,E2 -8415.778} C_VEL
LIN {X 0,Y 453.497,Z 426.992,A -85,B 0,C 180,E1 -8419.409,E2 -8419.409} C_VEL
LIN {X 0,Y 453.453,Z 427,A -85,B 0,C 180,E1 -8422.81,E2 -8422.81} C_VEL
LIN {X 0,Y 453.479,Z 426.995,A -85,B 0,C 180,E1 -8426.087,E2 -8426.087} C_VEL
LIN {X 0,Y 453.478,Z 426.994,A -85,B 0,C 180,E1 -8429.24,E2 -8429.24} C_VEL
LIN {X 0,Y 453.478,Z 426.999,A -85,B 0,C 180,E1 -8432.294,E2 -8432.294} C_VEL
LIN {X 0,Y 453.473,Z 426.996,A -85,B 0,C 180,E1 -8435.263,E2 -8435.263} C_VEL
LIN {X 0,Y 453.478,Z 427,A -85,B 0,C 180,E1 -8438.417,E2 -8438.417} C_VEL
LIN {X 0,Y 453.458,Z 427.002,A -85,B 0,C 180,E1 -8441.942,E2 -8441.942} C_VEL
LIN {X 0,Y 453.488,Z 426.996,A -85,B 0,C 180,E1 -8444.724,E2 -8444.724} C_VEL
LIN {X 0,Y 453.568,Z 426.986,A -85,B 0,C 180,E1 -8447.471,E2 -8447.471} C_VEL
LIN {X 0,Y 453.558,Z 426.988,A -85,B 0,C 180,E1 -8451.086,E2 -8451.086} C_VEL
LIN {X 0,Y 453.631,Z 426.982,A -85,B 0,C 180,E1 -8453.774,E2 -8453.774} C_VEL
LIN {X 0,Y 453.5,Z 427.18,A -85,B 0,C 180,E1 -8456.335,E2 -8456.335} C_VEL
LIN {X 0,Y 454.509,Z 431.109,A -85,B 0,C 180,E1 -8457.437,E2 -8457.437} C_VEL
LIN {X 0,Y 457.61,Z 440.742,A -85,B 0,C 180,E1 -8457.765,E2 -8457.765} C_VEL
LIN {X 0,Y 458.109,Z 443.938,A -85,B 0,C 180,E1 -8457.849,E2 -8457.849} C_VEL
LIN {X 0,Y 456.747,Z 537.5,A -85,B 0,C 180,E1 -8459.545,E2 -8459.545} C_VEL
LIN {X 0,Y 456.508,Z 550.649,A -85,B 0,C 180,E1 -8459.97,E2 -8459.97} C_VEL
LIN {X 0,Y 456.203,Z 563.015,A -85,B 0,C 180,E1 -8460.552,E2 -8460.552} C_VEL
LIN {X 0,Y 455.739,Z 575.243,A -85,B 0,C 180,E1 -8461.325,E2 -8461.325} C_VEL
LIN {X 0,Y 455.16,Z 586.255,A -85,B 0,C 180,E1 -8462.212,E2 -8462.212} C_VEL
LIN {X 0,Y 454.709,Z 595.162,A -85,B 0,C 180,E1 -8463.101,E2 -8463.101} C_VEL
LIN {X 0,Y 454.269,Z 604.321,A -85,B 0,C 180,E1 -8464.214,E2 -8464.214} C_VEL
LIN {X 0,Y 453.818,Z 613.22,A -85,B 0,C 180,E1 -8465.554,E2 -8465.554} C_VEL
LIN {X 0,Y 453.466,Z 620.86,A -85,B 0,C 180,E1 -8467.001,E2 -8467.001} C_VEL
LIN {X 0,Y 453.134,Z 626.892,A -85,B 0,C 180,E1 -8468.473,E2 -8468.473} C_VEL
LIN {X 0,Y 452.935,Z 631.172,A -85,B 0,C 180,E1 -8469.827,E2 -8469.827} C_VEL
LIN {X 0,Y 452.841,Z 633.429,A -85,B 0,C 180,E1 -8470.733,E2 -8470.733} C_VEL
LIN {X 0,Y 452.698,Z 635.814,A -85,B 0,C 180,E1 -8472.023,E2 -8472.023} C_VEL
LIN {X 0,Y 452.574,Z 637.448,A -85,B 0,C 180,E1 -8473.47,E2 -8473.47} C_VEL
LIN {X 0,Y 452.545,Z 637.928,A -85,B 0,C 180,E1 -8474.388,E2 -8474.388} C_VEL
LIN {X 0,Y 452.568,Z 637.857,A -85,B 0,C 180,E1 -8475.674,E2 -8475.674} C_VEL
LIN {X 0,Y 452.578,Z 636.726,A -85,B 0,C 180,E1 -8477.16,E2 -8477.16} C_VEL
LIN {X 0,Y 452.705,Z 634.238,A -85,B 0,C 180,E1 -8478.737,E2 -8478.737} C_VEL
LIN {X 0,Y 452.882,Z 630.052,A -85,B 0,C 180,E1 -8480.436,E2 -8480.436} C_VEL
LIN {X 0,Y 453.052,Z 625.209,A -85,B 0,C 180,E1 -8481.858,E2 -8481.858} C_VEL
LIN {X 0,Y 453.37,Z 618.896,A -85,B 0,C 180,E1 -8483.284,E2 -8483.284} C_VEL
LIN {X 0,Y 453.761,Z 610.872,A -85,B 0,C 180,E1 -8484.72,E2 -8484.72} C_VEL
LIN {X 0,Y 454.172,Z 602.396,A -85,B 0,C 180,E1 -8485.94,E2 -8485.94} C_VEL
LIN {X 0,Y 454.65,Z 592.108,A -85,B 0,C 180,E1 -8487.13,E2 -8487.13} C_VEL
LIN {X 0,Y 455.201,Z 581.125,A -85,B 0,C 180,E1 -8488.15,E2 -8488.15} C_VEL
LIN {X 0,Y 455.594,Z 570.367,A -85,B 0,C 180,E1 -8488.946,E2 -8488.946} C_VEL
LIN {X 0,Y 456.084,Z 557.627,A -85,B 0,C 180,E1 -8489.672,E2 -8489.672} C_VEL
LIN {X 0,Y 456.395,Z 544.371,A -85,B 0,C 180,E1 -8490.222,E2 -8490.222} C_VEL
LIN {X 0,Y 456.592,Z 531.012,A -85,B 0,C 180,E1 -8490.575,E2 -8490.575} C_VEL
LIN {X 0,Y 457.647,Z 442.03,A -85,B 0,C 180,E1 -8492.114,E2 -8492.114} C_VEL
LIN {X 0,Y 455.105,Z 432.337,A -85,B 0,C 180,E1 -8492.382,E2 -8492.382} C_VEL
LIN {X 0,Y 453.716,Z 427.991,A -85,B 0,C 180,E1 -8492.539,E2 -8492.539} C_VEL
LIN {X 0,Y 453.503,Z 426.996,A -85,B 0,C 180,E1 -8492.847,E2 -8492.847} C_VEL
LIN {X 0,Y 453.449,Z 427.002,A -85,B 0,C 180,E1 -8496.083,E2 -8496.083} C_VEL
LIN {X 0,Y 453.444,Z 426.997,A -85,B 0,C 180,E1 -8499.455,E2 -8499.455} C_VEL
LIN {X 0,Y 453.451,Z 426.999,A -85,B 0,C 180,E1 -8501.931,E2 -8501.931} C_VEL
LIN {X 0,Y 453.483,Z 426.992,A -85,B 0,C 180,E1 -8505.471,E2 -8505.471} C_VEL
LIN {X 0,Y 453.472,Z 426.994,A -85,B 0,C 180,E1 -8509.388,E2 -8509.388} C_VEL
LIN {X 0,Y 453.438,Z 427.001,A -85,B 0,C 180,E1 -8512.808,E2 -8512.808} C_VEL
LIN {X 0,Y 453.477,Z 426.997,A -85,B 0,C 180,E1 -8516.087,E2 -8516.087} C_VEL
LIN {X 0,Y 453.476,Z 426.993,A -85,B 0,C 180,E1 -8519.24,E2 -8519.24} C_VEL
LIN {X 0,Y 453.491,Z 426.998,A -85,B 0,C 180,E1 -8522.294,E2 -8522.294} C_VEL
LIN {X 0,Y 453.479,Z 426.995,A -85,B 0,C 180,E1 -8524.636,E2 -8524.636} C_VEL
LIN {X 0,Y 452.807,Z 427.077,A -85,B 0,C 180,E1 -8525.377,E2 -8525.377} C_VEL
LIN {X 0,Y 449.952,Z 427.439,A -85,B 0,C 180,E1 -8526.581,E2 -8526.581} C_VEL
LIN {X 0,Y 447.548,Z 427.738,A -85,B 0,C 180,E1 -8527.551,E2 -8527.551} C_VEL
LIN {X 0,Y 446.526,Z 427.865,A -85,B 0,C 180,E1 -8528.301,E2 -8528.301} C_VEL
LIN {X 0,Y 446.449,Z 427.873,A -85,B 0,C 180,E1 -8528.555,E2 -8528.555} C_VEL
LIN {X 0,Y 446.449,Z 427.869,A -85,B 0,C 180,E1 -8531.648,E2 -8531.648} C_VEL
LIN {X 0,Y 446.495,Z 427.871,A -85,B 0,C 180,E1 -8534.479,E2 -8534.479} C_VEL
LIN {X 0,Y 446.519,Z 427.864,A -85,B 0,C 180,E1 -8538.193,E2 -8538.193} C_VEL
LIN {X 0,Y 446.533,Z 427.861,A -85,B 0,C 180,E1 -8540.944,E2 -8540.944} C_VEL
LIN {X 0,Y 446.614,Z 427.848,A -85,B 0,C 180,E1 -8543.676,E2 -8543.676} C_VEL
LIN {X 0,Y 446.683,Z 427.84,A -85,B 0,C 180,E1 -8547.294,E2 -8547.294} C_VEL
LIN {X 0,Y 446.789,Z 427.829,A -85,B 0,C 180,E1 -8550,E2 -8550} C_VEL
LIN {X 0,Y 446.679,Z 427.845,A -85,B 0,C 180,E1 -8552.705,E2 -8552.705} C_VEL
LIN {X 0,Y 446.641,Z 427.85,A -85,B 0,C 180,E1 -8556.323,E2 -8556.323} C_VEL
LIN {X 0,Y 446.533,Z 427.86,A -85,B 0,C 180,E1 -8559.055,E2 -8559.055} C_VEL
LIN {X 0,Y 446.523,Z 427.865,A -85,B 0,C 180,E1 -8562.729,E2 -8562.729} C_VEL
LIN {X 0,Y 446.497,Z 427.867,A -85,B 0,C 180,E1 -8566.227,E2 -8566.227} C_VEL
LIN {X 0,Y 446.469,Z 427.867,A -85,B 0,C 180,E1 -8569.303,E2 -8569.303} C_VEL
LIN {X 0,Y 446.419,Z 427.876,A -85,B 0,C 180,E1 -8572.199,E2 -8572.199} C_VEL
LIN {X 0,Y 446.442,Z 427.871,A -85,B 0,C 180,E1 -8575.153,E2 -8575.153} C_VEL
LIN {X 0,Y 446.449,Z 427.872,A -85,B 0,C 180,E1 -8578.181,E2 -8578.181} C_VEL
LIN {X 0,Y 446.416,Z 427.873,A -85,B 0,C 180,E1 -8581.3,E2 -8581.3} C_VEL
LIN {X 0,Y 446.429,Z 427.879,A -85,B 0,C 180,E1 -8584.523,E2 -8584.523} C_VEL
LIN {X 0,Y 446.41,Z 427.876,A -85,B 0,C 180,E1 -8588.078,E2 -8588.078} C_VEL
LIN {X 0,Y 446.418,Z 427.873,A -85,B 0,C 180,E1 -8591.392,E2 -8591.392} C_VEL
LIN {X 0,Y 446.449,Z 427.87,A -85,B 0,C 180,E1 -8595.104,E2 -8595.104} C_VEL
LIN {X 0,Y 446.418,Z 427.88,A -85,B 0,C 180,E1 -8598.608,E2 -8598.608} C_VEL
LIN {X 0,Y 446.436,Z 427.873,A -85,B 0,C 180,E1 -8600.972,E2 -8600.972} C_VEL
LIN {X 0,Y 446.416,Z 427.878,A -85,B 0,C 180,E1 -8604.374,E2 -8604.374} C_VEL
LIN {X 0,Y 446.422,Z 427.872,A -85,B 0,C 180,E1 -8607.638,E2 -8607.638} C_VEL
LIN {X 0,Y 446.447,Z 427.874,A -85,B 0,C 180,E1 -8610.79,E2 -8610.79} C_VEL
LIN {X 0,Y 446.459,Z 427.868,A -85,B 0,C 180,E1 -8613.847,E2 -8613.847} C_VEL
LIN {X 0,Y 446.425,Z 427.877,A -85,B 0,C 180,E1 -8616.823,E2 -8616.823} C_VEL
LIN {X 0,Y 446.443,Z 427.869,A -85,B 0,C 180,E1 -8619.737,E2 -8619.737} C_VEL
LIN {X 0,Y 446.456,Z 427.876,A -85,B 0,C 180,E1 -8622.597,E2 -8622.597} C_VEL
LIN {X 0,Y 446.469,Z 427.867,A -85,B 0,C 180,E1 -8625.412,E2 -8625.412} C_VEL
LIN {X 0,Y 446.517,Z 427.863,A -85,B 0,C 180,E1 -8628.193,E2 -8628.193} C_VEL
LIN {X 0,Y 446.536,Z 427.862,A -85,B 0,C 180,E1 -8630.945,E2 -8630.945} C_VEL
LIN {X 0,Y 446.621,Z 427.847,A -85,B 0,C 180,E1 -8633.676,E2 -8633.676} C_VEL
LIN {X 0,Y 446.69,Z 427.84,A -85,B 0,C 180,E1 -8637.295,E2 -8637.295} C_VEL
LIN {X 0,Y 446.792,Z 427.827,A -85,B 0,C 180,E1 -8640,E2 -8640} C_VEL
LIN {X 0,Y 446.706,Z 427.844,A -85,B 0,C 180,E1 -8642.705,E2 -8642.705} C_VEL
LIN {X 0,Y 446.646,Z 427.848,A -85,B 0,C 180,E1 -8646.324,E2 -8646.324} C_VEL
LIN {X 0,Y 446.536,Z 427.861,A -85,B 0,C 180,E1 -8649.055,E2 -8649.055} C_VEL
LIN {X 0,Y 446.521,Z 427.867,A -85,B 0,C 180,E1 -8652.73,E2 -8652.73} C_VEL
LIN {X 0,Y 446.495,Z 427.865,A -85,B 0,C 180,E1 -8656.228,E2 -8656.228} C_VEL
LIN {X 0,Y 446.468,Z 427.867,A -85,B 0,C 180,E1 -8659.303,E2 -8659.303} C_VEL
LIN {X 0,Y 446.418,Z 427.875,A -85,B 0,C 180,E1 -8662.2,E2 -8662.2} C_VEL
LIN {X 0,Y 446.444,Z 427.872,A -85,B 0,C 180,E1 -8665.153,E2 -8665.153} C_VEL
LIN {X 0,Y 446.484,Z 427.866,A -85,B 0,C 180,E1 -8668.179,E2 -8668.179} C_VEL
LIN {X 0,Y 446.419,Z 427.872,A -85,B 0,C 180,E1 -8671.775,E2 -8671.775} C_VEL
LIN {X 0,Y 446.429,Z 427.877,A -85,B 0,C 180,E1 -8674.523,E2 -8674.523} C_VEL
LIN {X 0,Y 446.415,Z 427.874,A -85,B 0,C 180,E1 -8678.079,E2 -8678.079} C_VEL
LIN {X 0,Y 446.427,Z 427.877,A -85,B 0,C 180,E1 -8680.918,E2 -8680.918} C_VEL
LIN {X 0,Y 446.402,Z 427.875,A -85,B 0,C 180,E1 -8683.846,E2 -8683.846} C_VEL
LIN {X 0,Y 446.421,Z 427.876,A -85,B 0,C 180,E1 -8686.401,E2 -8686.401} C_VEL
LIN {X 0,Y 446.448,Z 427.869,A -85,B 0,C 180,E1 -8689.803,E2 -8689.803} C_VEL
LIN {X 0,Y 446.408,Z 427.875,A -85,B 0,C 180,E1 -8692.121,E2 -8692.121} C_VEL
LIN {X 0,Y 446.429,Z 427.872,A -85,B 0,C 180,E1 -8695.477,E2 -8695.477} C_VEL
LIN {X 0,Y 446.417,Z 427.878,A -85,B 0,C 180,E1 -8698.7,E2 -8698.7} C_VEL
LIN {X 0,Y 446.515,Z 427.901,A -85,B 0,C 180,E1 -8701.279,E2 -8701.279} C_VEL
LIN {X 0,Y 449.623,Z 443.074,A -85,B 0,C 180,E1 -8704.045,E2 -8704.045} C_VEL
LIN {X 0,Y 449.628,Z 448.949,A -85,B 0,C 180,E1 -8705.038,E2 -8705.038} C_VEL
LIN {X 0,Y 448.504,Z 469.326,A -85,B 0,C 180,E1 -8708.393,E2 -8708.393} C_VEL
LIN {X 0,Y 447.571,Z 489.658,A -85,B 0,C 180,E1 -8711.697,E2 -8711.697} C_VEL
LIN {X 0,Y 447.423,Z 492.97,A -85,B 0,C 180,E1 -8712.232,E2 -8712.232} C_VEL
LIN {X 0,Y 450.495,Z 516.693,A -85,B 0,C 180,E1 -8712.779,E2 -8712.779} C_VEL
LIN {X 0,Y 449.474,Z 603.284,A -85,B 0,C 180,E1 -8714.324,E2 -8714.324} C_VEL
LIN {X 0,Y 449.059,Z 615.837,A -85,B 0,C 180,E1 -8714.716,E2 -8714.716} C_VEL
LIN {X 0,Y 448.458,Z 628.794,A -85,B 0,C 180,E1 -8715.305,E2 -8715.305} C_VEL
LIN {X 0,Y 447.965,Z 640.651,A -85,B 0,C 180,E1 -8716.042,E2 -8716.042} C_VEL
LIN {X 0,Y 447.376,Z 652.353,A -85,B 0,C 180,E1 -8716.971,E2 -8716.971} C_VEL
LIN {X 0,Y 446.791,Z 662.452,A -85,B 0,C 180,E1 -8717.97,E2 -8717.97} C_VEL
LIN {X 0,Y 446.411,Z 671.768,A -85,B 0,C 180,E1 -8719.111,E2 -8719.111} C_VEL
LIN {X 0,Y 446.002,Z 680.835,A -85,B 0,C 180,E1 -8720.477,E2 -8720.477} C_VEL
LIN {X 0,Y 445.757,Z 688.116,A -85,B 0,C 180,E1 -8721.843,E2 -8721.843} C_VEL
LIN {X 0,Y 445.593,Z 694.064,A -85,B 0,C 180,E1 -8723.252,E2 -8723.252} C_VEL
LIN {X 0,Y 445.553,Z 698.437,A -85,B 0,C 180,E1 -8724.57,E2 -8724.57} C_VEL
LIN {X 0,Y 445.45,Z 700.814,A -85,B 0,C 180,E1 -8725.476,E2 -8725.476} C_VEL
LIN {X 0,Y 445.517,Z 702.759,A -85,B 0,C 180,E1 -8726.383,E2 -8726.383} C_VEL
LIN {X 0,Y 445.529,Z 704.233,A -85,B 0,C 180,E1 -8727.288,E2 -8727.288} C_VEL
LIN {X 0,Y 445.518,Z 705.255,A -85,B 0,C 180,E1 -8728.192,E2 -8728.192} C_VEL
LIN {X 0,Y 445.438,Z 705.864,A -85,B 0,C 180,E1 -8729.096,E2 -8729.096} C_VEL
LIN {X 0,Y 445.421,Z 706.071,A -85,B 0,C 180,E1 -8730,E2 -8730} C_VEL
LIN {X 0,Y 445.439,Z 705.831,A -85,B 0,C 180,E1 -8730.904,E2 -8730.904} C_VEL
LIN {X 0,Y 445.52,Z 705.172,A -85,B 0,C 180,E1 -8731.808,E2 -8731.808} C_VEL
LIN {X 0,Y 445.543,Z 704.103,A -85,B 0,C 180,E1 -8732.713,E2 -8732.713} C_VEL
LIN {X 0,Y 445.529,Z 702.608,A -85,B 0,C 180,E1 -8733.618,E2 -8733.618} C_VEL
LIN {X 0,Y 445.511,Z 699.488,A -85,B 0,C 180,E1 -8734.978,E2 -8734.978} C_VEL
LIN {X 0,Y 445.548,Z 695.044,A -85,B 0,C 180,E1 -8736.406,E2 -8736.406} C_VEL
LIN {X 0,Y 445.715,Z 688.826,A -85,B 0,C 180,E1 -8737.931,E2 -8737.931} C_VEL
LIN {X 0,Y 445.943,Z 681.791,A -85,B 0,C 180,E1 -8739.297,E2 -8739.297} C_VEL
LIN {X 0,Y 446.314,Z 673.062,A -85,B 0,C 180,E1 -8740.663,E2 -8740.663} C_VEL
LIN {X 0,Y 446.688,Z 663.06,A -85,B 0,C 180,E1 -8741.918,E2 -8741.918} C_VEL
LIN {X 0,Y 447.321,Z 652.563,A -85,B 0,C 180,E1 -8742.986,E2 -8742.986} C_VEL
LIN {X 0,Y 447.831,Z 642.14,A -85,B 0,C 180,E1 -8743.847,E2 -8743.847} C_VEL
LIN {X 0,Y 448.443,Z 629.951,A -85,B 0,C 180,E1 -8744.638,E2 -8744.638} C_VEL
LIN {X 0,Y 449.058,Z 617.369,A -85,B 0,C 180,E1 -8745.256,E2 -8745.256} C_VEL
LIN {X 0,Y 449.557,Z 604.37,A -85,B 0,C 180,E1 -8745.703,E2 -8745.703} C_VEL
LIN {X 0,Y 449.878,Z 586.319,A -85,B 0,C 180,E1 -8746.07,E2 -8746.07} C_VEL
LIN {X 0,Y 450.612,Z 515.586,A -85,B 0,C 180,E1 -8747.355,E2 -8747.355} C_VEL
LIN {X 0,Y 447.583,Z 491.922,A -85,B 0,C 180,E1 -8747.951,E2 -8747.951} C_VEL
LIN {X 0,Y 447.367,Z 490.113,A -85,B 0,C 180,E1 -8748.019,E2 -8748.019} C_VEL
LIN {X 0,Y 448.185,Z 471.065,A -85,B 0,C 180,E1 -8751.141,E2 -8751.141} C_VEL
LIN {X 0,Y 449.149,Z 453.913,A -85,B 0,C 180,E1 -8754.006,E2 -8754.006} C_VEL
LIN {X 0,Y 449.687,Z 443.977,A -85,B 0,C 180,E1 -8755.703,E2 -8755.703} C_VEL
LIN {X 0,Y 447.932,Z 434.108,A -85,B 0,C 180,E1 -8757.572,E2 -8757.572} C_VEL
LIN {X 0,Y 446.486,Z 427.872,A -85,B 0,C 180,E1 -8758.82,E2 -8758.82} C_VEL
LIN {X 0,Y 446.426,Z 427.882,A -85,B 0,C 180,E1 -8762.362,E2 -8762.362} C_VEL
LIN {X 0,Y 446.423,Z 427.879,A -85,B 0,C 180,E1 -8765.626,E2 -8765.626} C_VEL
LIN {X 0,Y 446.459,Z 427.874,A -85,B 0,C 180,E1 -8769.026,E2 -8769.026} C_VEL
LIN {X 0,Y 446.438,Z 427.875,A -85,B 0,C 180,E1 -8772.278,E2 -8772.278} C_VEL
LIN {X 0,Y 446.454,Z 427.872,A -85,B 0,C 180,E1 -8775.104,E2 -8775.104} C_VEL
LIN {X 0,Y 446.422,Z 427.88,A -85,B 0,C 180,E1 -8778.608,E2 -8778.608} C_VEL
LIN {X 0,Y 446.428,Z 427.875,A -85,B 0,C 180,E1 -8780.971,E2 -8780.971} C_VEL
LIN {X 0,Y 446.421,Z 427.878,A -85,B 0,C 180,E1 -8784.374,E2 -8784.374} C_VEL
LIN {X 0,Y 446.425,Z 427.872,A -85,B 0,C 180,E1 -8787.639,E2 -8787.639} C_VEL
LIN {X 0,Y 446.425,Z 427.876,A -85,B 0,C 180,E1 -8790.789,E2 -8790.789} C_VEL
LIN {X 0,Y 446.439,Z 427.874,A -85,B 0,C 180,E1 -8793.846,E2 -8793.846} C_VEL
LIN {X 0,Y 446.426,Z 427.875,A -85,B 0,C 180,E1 -8796.823,E2 -8796.823} C_VEL
LIN {X 0,Y 446.391,Z 427.88,A -85,B 0,C 180,E1 -8799.734,E2 -8799.734} C_VEL
LIN {X 0,Y 446.391,Z 427.88,A -85,B 0,C 180,E1 -8802.594,E2 -8802.594} C_VEL
LIN {X 0,Y 446.436,Z 427.875,A -85,B 0,C 180,E1 -8805.411,E2 -8805.411} C_VEL
LIN {X 0,Y 446.506,Z 427.869,A -85,B 0,C 180,E1 -8808.193,E2 -8808.193} C_VEL
LIN {X 0,Y 446.508,Z 427.866,A -85,B 0,C 180,E1 -8810.944,E2 -8810.944} C_VEL
LIN {X 0,Y 446.602,Z 427.858,A -85,B 0,C 180,E1 -8813.676,E2 -8813.676} C_VEL
LIN {X 0,Y 446.442,Z 427.912,A -85,B 0,C 180,E1 -8815.994,E2 -8815.994} C_VEL
LIN {X 0,Y 447.364,Z 431.854,A -85,B 0,C 180,E1 -8817.101,E2 -8817.101} C_VEL
LIN {X 0,Y 450.47,Z 440.316,A -85,B 0,C 180,E1 -8817.423,E2 -8817.423} C_VEL
LIN {X 0,Y 451.447,Z 444.308,A -85,B 0,C 180,E1 -8817.549,E2 -8817.549} C_VEL
LIN {X 0,Y 449.965,Z 537.564,A -85,B 0,C 180,E1 -8819.281,E2 -8819.281} C_VEL
LIN {X 0,Y 449.709,Z 551.135,A -85,B 0,C 180,E1 -8819.723,E2 -8819.723} C_VEL
LIN {X 0,Y 449.396,Z 562.952,A -85,B 0,C 180,E1 -8820.28,E2 -8820.28} C_VEL
LIN {X 0,Y 448.928,Z 574.56,A -85,B 0,C 180,E1 -8821.009,E2 -8821.009} C_VEL
LIN {X 0,Y 448.347,Z 585.791,A -85,B 0,C 180,E1 -8821.909,E2 -8821.909} C_VEL
LIN {X 0,Y 447.811,Z 595.935,A -85,B 0,C 180,E1 -8822.924,E2 -8822.924} C_VEL
LIN {X 0,Y 447.328,Z 605.045,A -85,B 0,C 180,E1 -8824.054,E2 -8824.054} C_VEL
LIN {X 0,Y 446.834,Z 613.906,A -85,B 0,C 180,E1 -8825.415,E2 -8825.415} C_VEL
LIN {X 0,Y 446.497,Z 621.028,A -85,B 0,C 180,E1 -8826.78,E2 -8826.78} C_VEL
LIN {X 0,Y 446.154,Z 626.711,A -85,B 0,C 180,E1 -8828.15,E2 -8828.15} C_VEL
LIN {X 0,Y 445.929,Z 631.164,A -85,B 0,C 180,E1 -8829.525,E2 -8829.525} C_VEL
LIN {X 0,Y 445.745,Z 634.516,A -85,B 0,C 180,E1 -8830.906,E2 -8830.906} C_VEL
LIN {X 0,Y 445.634,Z 636.579,A -85,B 0,C 180,E1 -8832.096,E2 -8832.096} C_VEL
LIN {X 0,Y 445.484,Z 638.178,A -85,B 0,C 180,E1 -8833.688,E2 -8833.688} C_VEL
LIN {X 0,Y 445.482,Z 638.508,A -85,B 0,C 180,E1 -8834.621,E2 -8834.621} C_VEL
LIN {X 0,Y 445.497,Z 638.355,A -85,B 0,C 180,E1 -8835.778,E2 -8835.778} C_VEL
LIN {X 0,Y 445.511,Z 636.919,A -85,B 0,C 180,E1 -8837.441,E2 -8837.441} C_VEL
LIN {X 0,Y 445.654,Z 634.555,A -85,B 0,C 180,E1 -8838.877,E2 -8838.877} C_VEL
LIN {X 0,Y 445.802,Z 631.143,A -85,B 0,C 180,E1 -8840.293,E2 -8840.293} C_VEL
LIN {X 0,Y 445.984,Z 626.158,A -85,B 0,C 180,E1 -8841.819,E2 -8841.819} C_VEL
LIN {X 0,Y 446.281,Z 620.387,A -85,B 0,C 180,E1 -8843.185,E2 -8843.185} C_VEL
LIN {X 0,Y 446.678,Z 612.581,A -85,B 0,C 180,E1 -8844.642,E2 -8844.642} C_VEL
LIN {X 0,Y 447.097,Z 604.483,A -85,B 0,C 180,E1 -8845.862,E2 -8845.862} C_VEL
LIN {X 0,Y 447.601,Z 594.486,A -85,B 0,C 180,E1 -8847.087,E2 -8847.087} C_VEL
LIN {X 0,Y 448.068,Z 584.505,A -85,B 0,C 180,E1 -8848.07,E2 -8848.07} C_VEL
LIN {X 0,Y 448.58,Z 573.791,A -85,B 0,C 180,E1 -8848.923,E2 -8848.923} C_VEL
LIN {X 0,Y 449.037,Z 561.951,A -85,B 0,C 180,E1 -8849.668,E2 -8849.668} C_VEL
LIN {X 0,Y 449.429,Z 549.15,A -85,B 0,C 180,E1 -8850.264,E2 -8850.264} C_VEL
LIN {X 0,Y 449.713,Z 535.452,A -85,B 0,C 180,E1 -8850.696,E2 -8850.696} C_VEL
LIN {X 0,Y 450.777,Z 442.847,A -85,B 0,C 180,E1 -8852.351,E2 -8852.351} C_VEL
LIN {X 0,Y 448.06,Z 433.15,A -85,B 0,C 180,E1 -8852.632,E2 -8852.632} C_VEL
LIN {X 0,Y 446.584,Z 428.487,A -85,B 0,C 180,E1 -8852.788,E2 -8852.788} C_VEL
LIN {X 0,Y 446.476,Z 427.87,A -85,B 0,C 180,E1 -8853.008,E2 -8853.008} C_VEL
LIN {X 0,Y 446.416,Z 427.875,A -85,B 0,C 180,E1 -8855.626,E2 -8855.626} C_VEL
LIN {X 0,Y 446.402,Z 427.876,A -85,B 0,C 180,E1 -8859.031,E2 -8859.031} C_VEL
LIN {X 0,Y 446.394,Z 427.882,A -85,B 0,C 180,E1 -8862.271,E2 -8862.271} C_VEL
LIN {X 0,Y 446.424,Z 427.872,A -85,B 0,C 180,E1 -8865.107,E2 -8865.107} C_VEL
LIN {X 0,Y 446.403,Z 427.88,A -85,B 0,C 180,E1 -8868.605,E2 -8868.605} C_VEL
LIN {X 0,Y 446.4,Z 427.877,A -85,B 0,C 180,E1 -8871.923,E2 -8871.923} C_VEL
LIN {X 0,Y 446.428,Z 427.871,A -85,B 0,C 180,E1 -8875.476,E2 -8875.476} C_VEL
LIN {X 0,Y 446.417,Z 427.877,A -85,B 0,C 180,E1 -8878.699,E2 -8878.699} C_VEL
LIN {X 0,Y 446.449,Z 427.87,A -85,B 0,C 180,E1 -8881.83,E2 -8881.83} C_VEL
LIN {X 0,Y 446.434,Z 427.873,A -85,B 0,C 180,E1 -8884.846,E2 -8884.846} C_VEL
LIN {X 0,Y 446.451,Z 427.874,A -85,B 0,C 180,E1 -8888.245,E2 -8888.245} C_VEL
LIN {X 0,Y 446.449,Z 427.873,A -85,B 0,C 180,E1 -8888.555,E2 -8888.555} C_VEL
LIN {X 0,Y 445.793,Z 427.955,A -85,B 0,C 180,E1 -8889.309,E2 -8889.309} C_VEL
LIN {X 0,Y 442.933,Z 428.315,A -85,B 0,C 180,E1 -8890.532,E2 -8890.532} C_VEL
LIN {X 0,Y 440.511,Z 428.618,A -85,B 0,C 180,E1 -8891.52,E2 -8891.52} C_VEL
LIN {X 0,Y 439.48,Z 428.743,A -85,B 0,C 180,E1 -8892.283,E2 -8892.283} C_VEL
LIN {X 0,Y 439.401,Z 428.75,A -85,B 0,C 180,E1 -8892.541,E2 -8892.541} C_VEL
LIN {X 0,Y 439.442,Z 428.742,A -85,B 0,C 180,E1 -8895.173,E2 -8895.173} C_VEL
LIN {X 0,Y 439.485,Z 428.739,A -85,B 0,C 180,E1 -8898.001,E2 -8898.001} C_VEL
LIN {X 0,Y 439.505,Z 428.734,A -85,B 0,C 180,E1 -8901.725,E2 -8901.725} C_VEL
LIN {X 0,Y 439.606,Z 428.729,A -85,B 0,C 180,E1 -8904.495,E2 -8904.495} C_VEL
LIN {X 0,Y 439.634,Z 428.721,A -85,B 0,C 180,E1 -8908.167,E2 -8908.167} C_VEL
LIN {X 0,Y 439.758,Z 428.704,A -85,B 0,C 180,E1 -8910,E2 -8910} C_VEL
LIN {X 0,Y 439.628,Z 428.723,A -85,B 0,C 180,E1 -8912.749,E2 -8912.749} C_VEL
LIN {X 0,Y 439.61,Z 428.728,A -85,B 0,C 180,E1 -8916.425,E2 -8916.425} C_VEL
LIN {X 0,Y 439.496,Z 428.736,A -85,B 0,C 180,E1 -8919.201,E2 -8919.201} C_VEL
LIN {X 0,Y 439.467,Z 428.741,A -85,B 0,C 180,E1 -8922.937,E2 -8922.937} C_VEL
LIN {X 0,Y 439.447,Z 428.747,A -85,B 0,C 180,E1 -8926.348,E2 -8926.348} C_VEL
LIN {X 0,Y 439.403,Z 428.746,A -85,B 0,C 180,E1 -8929.626,E2 -8929.626} C_VEL
LIN {X 0,Y 439.364,Z 428.759,A -85,B 0,C 180,E1 -8932.575,E2 -8932.575} C_VEL
LIN {X 0,Y 439.38,Z 428.749,A -85,B 0,C 180,E1 -8935.586,E2 -8935.586} C_VEL
LIN {X 0,Y 439.4,Z 428.753,A -85,B 0,C 180,E1 -8938.674,E2 -8938.674} C_VEL
LIN {X 0,Y 439.37,Z 428.752,A -85,B 0,C 180,E1 -8942.03,E2 -8942.03} C_VEL
LIN {X 0,Y 439.393,Z 428.748,A -85,B 0,C 180,E1 -8945.34,E2 -8945.34} C_VEL
LIN {X 0,Y 439.362,Z 428.759,A -85,B 0,C 180,E1 -8948.597,E2 -8948.597} C_VEL
LIN {X 0,Y 439.38,Z 428.75,A -85,B 0,C 180,E1 -8951.255,E2 -8951.255} C_VEL
LIN {X 0,Y 439.397,Z 428.753,A -85,B 0,C 180,E1 -8954.729,E2 -8954.729} C_VEL
LIN {X 0,Y 439.383,Z 428.749,A -85,B 0,C 180,E1 -8957.794,E2 -8957.794} C_VEL
LIN {X 0,Y 439.392,Z 428.751,A -85,B 0,C 180,E1 -8960.224,E2 -8960.224} C_VEL
LIN {X 0,Y 439.371,Z 428.75,A -85,B 0,C 180,E1 -8963.712,E2 -8963.712} C_VEL
LIN {X 0,Y 439.372,Z 428.753,A -85,B 0,C 180,E1 -8967.054,E2 -8967.054} C_VEL
LIN {X 0,Y 439.381,Z 428.753,A -85,B 0,C 180,E1 -8970.274,E2 -8970.274} C_VEL
LIN {X 0,Y 439.418,Z 428.745,A -85,B 0,C 180,E1 -8973.396,E2 -8973.396} C_VEL
LIN {X 0,Y 439.383,Z 428.754,A -85,B 0,C 180,E1 -8976.429,E2 -8976.429} C_VEL
LIN {X 0,Y 439.387,Z 428.749,A -85,B 0,C 180,E1 -8979.397,E2 -8979.397} C_VEL
LIN {X 0,Y 439.405,Z 428.75,A -85,B 0,C 180,E1 -8982.308,E2 -8982.308} C_VEL
LIN {X 0,Y 439.446,Z 428.743,A -85,B 0,C 180,E1 -8985.174,E2 -8985.174} C_VEL
LIN {X 0,Y 439.483,Z 428.738,A -85,B 0,C 180,E1 -8988.001,E2 -8988.001} C_VEL
LIN {X 0,Y 439.532,Z 428.73,A -85,B 0,C 180,E1 -8991.726,E2 -8991.726} C_VEL
LIN {X 0,Y 439.61,Z 428.727,A -85,B 0,C 180,E1 -8994.496,E2 -8994.496} C_VEL
LIN {X 0,Y 439.635,Z 428.72,A -85,B 0,C 180,E1 -8998.168,E2 -8998.168} C_VEL
LIN {X 0,Y 439.762,Z 428.703,A -85,B 0,C 180,E1 -9000,E2 -9000} C_VEL
LIN {X 0,Y 439.653,Z 428.722,A -85,B 0,C 180,E1 -9002.749,E2 -9002.749} C_VEL
LIN {X 0,Y 439.618,Z 428.724,A -85,B 0,C 180,E1 -9006.425,E2 -9006.425} C_VEL
LIN {X 0,Y 439.498,Z 428.736,A -85,B 0,C 180,E1 -9009.202,E2 -9009.202} C_VEL
LIN {X 0,Y 439.466,Z 428.743,A -85,B 0,C 180,E1 -9012.938,E2 -9012.938} C_VEL
LIN {X 0,Y 439.446,Z 428.745,A -85,B 0,C 180,E1 -9016.348,E2 -9016.348} C_VEL
LIN {X 0,Y 439.402,Z 428.747,A -85,B 0,C 180,E1 -9019.626,E2 -9019.626} C_VEL
LIN {X 0,Y 439.364,Z 428.758,A -85,B 0,C 180,E1 -9022.576,E2 -9022.576} C_VEL
LIN {X 0,Y 439.389,Z 428.748,A -85,B 0,C 180,E1 -9025.586,E2 -9025.586} C_VEL
LIN {X 0,Y 439.417,Z 428.753,A -85,B 0,C 180,E1 -9028.674,E2 -9028.674} C_VEL
LIN {X 0,Y 439.37,Z 428.751,A -85,B 0,C 180,E1 -9032.031,E2 -9032.031} C_VEL
LIN {X 0,Y 439.394,Z 428.749,A -85,B 0,C 180,E1 -9035.341,E2 -9035.341} C_VEL
LIN {X 0,Y 439.377,Z 428.756,A -85,B 0,C 180,E1 -9038.596,E2 -9038.596} C_VEL
LIN {X 0,Y 439.388,Z 428.75,A -85,B 0,C 180,E1 -9041.257,E2 -9041.257} C_VEL
LIN {X 0,Y 439.402,Z 428.755,A -85,B 0,C 180,E1 -9044.729,E2 -9044.729} C_VEL
LIN {X 0,Y 439.397,Z 428.747,A -85,B 0,C 180,E1 -9047.796,E2 -9047.796} C_VEL
LIN {X 0,Y 439.43,Z 428.745,A -85,B 0,C 180,E1 -9050.228,E2 -9050.228} C_VEL
LIN {X 0,Y 439.372,Z 428.75,A -85,B 0,C 180,E1 -9053.713,E2 -9053.713} C_VEL
LIN {X 0,Y 439.373,Z 428.754,A -85,B 0,C 180,E1 -9057.054,E2 -9057.054} C_VEL
LIN {X 0,Y 439.443,Z 428.748,A -85,B 0,C 180,E1 -9060.936,E2 -9060.936} C_VEL
LIN {X 0,Y 439.455,Z 428.894,A -85,B 0,C 180,E1 -9061.068,E2 -9061.068} C_VEL
LIN {X 0,Y 442.627,Z 443.92,A -85,B 0,C 180,E1 -9063.857,E2 -9063.857} C_VEL
LIN {X 0,Y 442.762,Z 449.314,A -85,B 0,C 180,E1 -9064.792,E2 -9064.792} C_VEL
LIN {X 0,Y 441.512,Z 470.185,A -85,B 0,C 180,E1 -9068.279,E2 -9068.279} C_VEL
LIN {X 0,Y 440.532,Z 490.638,A -85,B 0,C 180,E1 -9071.659,E2 -9071.659} C_VEL
LIN {X 0,Y 440.443,Z 492.391,A -85,B 0,C 180,E1 -9071.947,E2 -9071.947} C_VEL
LIN {X 0,Y 443.64,Z 517.492,A -85,B 0,C 180,E1 -9072.556,E2 -9072.556} C_VEL
LIN {X 0,Y 442.572,Z 602.531,A -85,B 0,C 180,E1 -9074.102,E2 -9074.102} C_VEL
LIN {X 0,Y 442.12,Z 615.883,A -85,B 0,C 180,E1 -9074.529,E2 -9074.529} C_VEL
LIN {X 0,Y 441.501,Z 628.655,A -85,B 0,C 180,E1 -9075.127,E2 -9075.127} C_VEL
LIN {X 0,Y 440.945,Z 641.225,A -85,B 0,C 180,E1 -9075.933,E2 -9075.933} C_VEL
LIN {X 0,Y 440.348,Z 651.852,A -85,B 0,C 180,E1 -9076.798,E2 -9076.798} C_VEL
LIN {X 0,Y 439.833,Z 661.618,A -85,B 0,C 180,E1 -9077.777,E2 -9077.777} C_VEL
LIN {X 0,Y 439.374,Z 670.997,A -85,B 0,C 180,E1 -9078.934,E2 -9078.934} C_VEL
LIN {X 0,Y 438.949,Z 680.112,A -85,B 0,C 180,E1 -9080.322,E2 -9080.322} C_VEL
LIN {X 0,Y 438.68,Z 687.442,A -85,B 0,C 180,E1 -9081.71,E2 -9081.71} C_VEL
LIN {X 0,Y 438.515,Z 693.264,A -85,B 0,C 180,E1 -9083.097,E2 -9083.097} C_VEL
LIN {X 0,Y 438.467,Z 697.83,A -85,B 0,C 180,E1 -9084.482,E2 -9084.482} C_VEL
LIN {X 0,Y 438.377,Z 700.221,A -85,B 0,C 180,E1 -9085.403,E2 -9085.403} C_VEL
LIN {X 0,Y 438.421,Z 702.175,A -85,B 0,C 180,E1 -9086.324,E2 -9086.324} C_VEL
LIN {X 0,Y 438.452,Z 703.669,A -85,B 0,C 180,E1 -9087.244,E2 -9087.244} C_VEL
LIN {X 0,Y 438.46,Z 704.7,A -85,B 0,C 180,E1 -9088.163,E2 -9088.163} C_VEL
LIN {X 0,Y 438.377,Z 705.315,A -85,B 0,C 180,E1 -9089.082,E2 -9089.082} C_VEL
LIN {X 0,Y 438.358,Z 705.527,A -85,B 0,C 180,E1 -9090,E2 -9090} C_VEL
LIN {X 0,Y 438.378,Z 705.296,A -85,B 0,C 180,E1 -9090.919,E2 -9090.919} C_VEL
LIN {X 0,Y 438.462,Z 704.64,A -85,B 0,C 180,E1 -9091.837,E2 -9091.837} C_VEL
LIN {X 0,Y 438.466,Z 703.565,A -85,B 0,C 180,E1 -9092.757,E2 -9092.757} C_VEL
LIN {X 0,Y 438.431,Z 702.07,A -85,B 0,C 180,E1 -9093.677,E2 -9093.677} C_VEL
LIN {X 0,Y 438.445,Z 698.948,A -85,B 0,C 180,E1 -9095.058,E2 -9095.058} C_VEL
LIN {X 0,Y 438.468,Z 694.733,A -85,B 0,C 180,E1 -9096.442,E2 -9096.442} C_VEL
LIN {X 0,Y 438.662,Z 688.265,A -85,B 0,C 180,E1 -9098.059,E2 -9098.059} C_VEL
LIN {X 0,Y 438.879,Z 681.233,A -85,B 0,C 180,E1 -9099.448,E2 -9099.448} C_VEL
LIN {X 0,Y 439.302,Z 672.525,A -85,B 0,C 180,E1 -9100.835,E2 -9100.835} C_VEL
LIN {X 0,Y 439.724,Z 662.558,A -85,B 0,C 180,E1 -9102.109,E2 -9102.109} C_VEL
LIN {X 0,Y 440.38,Z 651.805,A -85,B 0,C 180,E1 -9103.22,E2 -9103.22} C_VEL
LIN {X 0,Y 441.019,Z 640.075,A -85,B 0,C 180,E1 -9104.183,E2 -9104.183} C_VEL
LIN {X 0,Y 441.64,Z 628.515,A -85,B 0,C 180,E1 -9104.928,E2 -9104.928} C_VEL
LIN {X 0,Y 442.24,Z 615.677,A -85,B 0,C 180,E1 -9105.556,E2 -9105.556} C_VEL
LIN {X 0,Y 442.773,Z 603.086,A -85,B 0,C 180,E1 -9105.98,E2 -9105.98} C_VEL
LIN {X 0,Y 443.042,Z 583.295,A -85,B 0,C 180,E1 -9106.384,E2 -9106.384} C_VEL
LIN {X 0,Y 443.984,Z 516.957,A -85,B 0,C 180,E1 -9107.62,E2 -9107.62} C_VEL
LIN {X 0,Y 440.969,Z 493.213,A -85,B 0,C 180,E1 -9108.236,E2 -9108.236} C_VEL
LIN {X 0,Y 440.438,Z 489.532,A -85,B 0,C 180,E1 -9108.346,E2 -9108.346} C_VEL
LIN {X 0,Y 441.216,Z 472.176,A -85,B 0,C 180,E1 -9111.247,E2 -9111.247} C_VEL
LIN {X 0,Y 442.13,Z 456.519,A -85,B 0,C 180,E1 -9113.913,E2 -9113.913} C_VEL
LIN {X 0,Y 442.815,Z 445.24,A -85,B 0,C 180,E1 -9115.879,E2 -9115.879} C_VEL
LIN {X 0,Y 440.981,Z 435.416,A -85,B 0,C 180,E1 -9117.786,E2 -9117.786} C_VEL
LIN {X 0,Y 439.428,Z 428.75,A -85,B 0,C 180,E1 -9119.197,E2 -9119.197} C_VEL
LIN {X 0,Y 439.376,Z 428.762,A -85,B 0,C 180,E1 -9122.946,E2 -9122.946} C_VEL
LIN {X 0,Y 439.377,Z 428.757,A -85,B 0,C 180,E1 -9126.287,E2 -9126.287} C_VEL
LIN {X 0,Y 439.41,Z 428.749,A -85,B 0,C 180,E1 -9129.85,E2 -9129.85} C_VEL
LIN {X 0,Y 439.385,Z 428.755,A -85,B 0,C 180,E1 -9132.627,E2 -9132.627} C_VEL
LIN {X 0,Y 439.402,Z 428.749,A -85,B 0,C 180,E1 -9135.271,E2 -9135.271} C_VEL
LIN {X 0,Y 439.385,Z 428.754,A -85,B 0,C 180,E1 -9138.745,E2 -9138.745} C_VEL
LIN {X 0,Y 439.372,Z 428.752,A -85,B 0,C 180,E1 -9141.609,E2 -9141.609} C_VEL
LIN {X 0,Y 439.402,Z 428.75,A -85,B 0,C 180,E1 -9144.844,E2 -9144.844} C_VEL
LIN {X 0,Y 439.376,Z 428.753,A -85,B 0,C 180,E1 -9148.14,E2 -9148.14} C_VEL
LIN {X 0,Y 439.403,Z 428.748,A -85,B 0,C 180,E1 -9151.606,E2 -9151.606} C_VEL
LIN {X 0,Y 439.37,Z 428.757,A -85,B 0,C 180,E1 -9154.413,E2 -9154.413} C_VEL
LIN {X 0,Y 439.364,Z 428.754,A -85,B 0,C 180,E1 -9157.424,E2 -9157.424} C_VEL
LIN {X 0,Y 439.384,Z 428.752,A -85,B 0,C 180,E1 -9160.686,E2 -9160.686} C_VEL
LIN {X 0,Y 439.404,Z 428.753,A -85,B 0,C 180,E1 -9164.222,E2 -9164.222} C_VEL
LIN {X 0,Y 439.469,Z 428.742,A -85,B 0,C 180,E1 -9167.297,E2 -9167.297} C_VEL
LIN {X 0,Y 439.475,Z 428.742,A -85,B 0,C 180,E1 -9170.798,E2 -9170.798} C_VEL
LIN {X 0,Y 439.553,Z 428.736,A -85,B 0,C 180,E1 -9173.574,E2 -9173.574} C_VEL
LIN {X 0,Y 439.415,Z 428.907,A -85,B 0,C 180,E1 -9175.7,E2 -9175.7} C_VEL
LIN {X 0,Y 440.201,Z 432.464,A -85,B 0,C 180,E1 -9176.739,E2 -9176.739} C_VEL
LIN {X 0,Y 444.081,Z 442.575,A -85,B 0,C 180,E1 -9177.154,E2 -9177.154} C_VEL
LIN {X 0,Y 444.794,Z 445.699,A -85,B 0,C 180,E1 -9177.252,E2 -9177.252} C_VEL
LIN {X 0,Y 443.183,Z 538.82,A -85,B 0,C 180,E1 -9179.036,E2 -9179.036} C_VEL
LIN {X 0,Y 442.906,Z 552.2,A -85,B 0,C 180,E1 -9179.487,E2 -9179.487} C_VEL
LIN {X 0,Y 442.576,Z 564.827,A -85,B 0,C 180,E1 -9180.114,E2 -9180.114} C_VEL
LIN {X 0,Y 442.008,Z 576.959,A -85,B 0,C 180,E1 -9180.911,E2 -9180.911} C_VEL
LIN {X 0,Y 441.401,Z 587.867,A -85,B 0,C 180,E1 -9181.825,E2 -9181.825} C_VEL
LIN {X 0,Y 440.848,Z 598.624,A -85,B 0,C 180,E1 -9182.97,E2 -9182.97} C_VEL
LIN {X 0,Y 440.278,Z 607.406,A -85,B 0,C 180,E1 -9184.119,E2 -9184.119} C_VEL
LIN {X 0,Y 439.805,Z 615.936,A -85,B 0,C 180,E1 -9185.502,E2 -9185.502} C_VEL
LIN {X 0,Y 439.491,Z 622.142,A -85,B 0,C 180,E1 -9186.752,E2 -9186.752} C_VEL
LIN {X 0,Y 439.068,Z 628.191,A -85,B 0,C 180,E1 -9188.283,E2 -9188.283} C_VEL
LIN {X 0,Y 438.849,Z 632.427,A -85,B 0,C 180,E1 -9189.68,E2 -9189.68} C_VEL
LIN {X 0,Y 438.663,Z 635.576,A -85,B 0,C 180,E1 -9191.084,E2 -9191.084} C_VEL
LIN {X 0,Y 438.559,Z 637.316,A -85,B 0,C 180,E1 -9192.164,E2 -9192.164} C_VEL
LIN {X 0,Y 438.418,Z 638.852,A -85,B 0,C 180,E1 -9193.913,E2 -9193.913} C_VEL
LIN {X 0,Y 438.404,Z 639.086,A -85,B 0,C 180,E1 -9194.862,E2 -9194.862} C_VEL
LIN {X 0,Y 438.423,Z 638.833,A -85,B 0,C 180,E1 -9195.884,E2 -9195.884} C_VEL
LIN {X 0,Y 438.419,Z 638.199,A -85,B 0,C 180,E1 -9196.771,E2 -9196.771} C_VEL
LIN {X 0,Y 438.449,Z 637.098,A -85,B 0,C 180,E1 -9197.731,E2 -9197.731} C_VEL
LIN {X 0,Y 438.595,Z 634.875,A -85,B 0,C 180,E1 -9199.018,E2 -9199.018} C_VEL
LIN {X 0,Y 438.768,Z 630.881,A -85,B 0,C 180,E1 -9200.633,E2 -9200.633} C_VEL
LIN {X 0,Y 438.984,Z 625.821,A -85,B 0,C 180,E1 -9202.126,E2 -9202.126} C_VEL
LIN {X 0,Y 439.313,Z 619.488,A -85,B 0,C 180,E1 -9203.575,E2 -9203.575} C_VEL
LIN {X 0,Y 439.778,Z 611.34,A -85,B 0,C 180,E1 -9205.055,E2 -9205.055} C_VEL
LIN {X 0,Y 440.235,Z 602.814,A -85,B 0,C 180,E1 -9206.296,E2 -9206.296} C_VEL
LIN {X 0,Y 440.771,Z 592.198,A -85,B 0,C 180,E1 -9207.542,E2 -9207.542} C_VEL
LIN {X 0,Y 441.338,Z 581.633,A -85,B 0,C 180,E1 -9208.537,E2 -9208.537} C_VEL
LIN {X 0,Y 441.828,Z 569.343,A -85,B 0,C 180,E1 -9209.448,E2 -9209.448} C_VEL
LIN {X 0,Y 442.338,Z 556.673,A -85,B 0,C 180,E1 -9210.163,E2 -9210.163} C_VEL
LIN {X 0,Y 442.655,Z 543.613,A -85,B 0,C 180,E1 -9210.689,E2 -9210.689} C_VEL
LIN {X 0,Y 442.87,Z 529.666,A -85,B 0,C 180,E1 -9211.046,E2 -9211.046} C_VEL
LIN {X 0,Y 444,Z 444.077,A -85,B 0,C 180,E1 -9212.581,E2 -9212.581} C_VEL
LIN {X 0,Y 441.317,Z 434.837,A -85,B 0,C 180,E1 -9212.858,E2 -9212.858} C_VEL
LIN {X 0,Y 439.48,Z 428.946,A -85,B 0,C 180,E1 -9213.056,E2 -9213.056} C_VEL
LIN {X 0,Y 439.371,Z 428.757,A -85,B 0,C 180,E1 -9216.288,E2 -9216.288} C_VEL
LIN {X 0,Y 439.361,Z 428.753,A -85,B 0,C 180,E1 -9219.78,E2 -9219.78} C_VEL
LIN {X 0,Y 439.346,Z 428.759,A -85,B 0,C 180,E1 -9222.621,E2 -9222.621} C_VEL
LIN {X 0,Y 439.378,Z 428.75,A -85,B 0,C 180,E1 -9225.267,E2 -9225.267} C_VEL
LIN {X 0,Y 439.365,Z 428.755,A -85,B 0,C 180,E1 -9228.747,E2 -9228.747} C_VEL
LIN {X 0,Y 439.358,Z 428.752,A -85,B 0,C 180,E1 -9231.611,E2 -9231.611} C_VEL
LIN {X 0,Y 439.397,Z 428.75,A -85,B 0,C 180,E1 -9234.843,E2 -9234.843} C_VEL
LIN {X 0,Y 439.375,Z 428.754,A -85,B 0,C 180,E1 -9238.139,E2 -9238.139} C_VEL
LIN {X 0,Y 439.402,Z 428.747,A -85,B 0,C 180,E1 -9241.606,E2 -9241.606} C_VEL
LIN {X 0,Y 439.375,Z 428.758,A -85,B 0,C 180,E1 -9244.413,E2 -9244.413} C_VEL
LIN {X 0,Y 439.365,Z 428.751,A -85,B 0,C 180,E1 -9247.424,E2 -9247.424} C_VEL
LIN {X 0,Y 439.443,Z 428.747,A -85,B 0,C 180,E1 -9250.663,E2 -9250.663} C_VEL
LIN {X 0,Y 439.401,Z 428.75,A -85,B 0,C 180,E1 -9252.541,E2 -9252.541} C_VEL
LIN {X 0,Y 438.742,Z 428.83,A -85,B 0,C 180,E1 -9253.306,E2 -9253.306} C_VEL
LIN {X 0,Y 435.873,Z 429.193,A -85,B 0,C 180,E1 -9254.549,E2 -9254.549} C_VEL
LIN {X 0,Y 433.458,Z 429.49,A -85,B 0,C 180,E1 -9255.552,E2 -9255.552} C_VEL
LIN {X 0,Y 432.448,Z 429.619,A -85,B 0,C 180,E1 -9256.328,E2 -9256.328} C_VEL
LIN {X 0,Y 432.381,Z 429.622,A -85,B 0,C 180,E1 -9256.59,E2 -9256.59} C_VEL
LIN {X 0,Y 432.391,Z 429.624,A -85,B 0,C 180,E1 -9258.752,E2 -9258.752} C_VEL
LIN {X 0,Y 432.465,Z 429.611,A -85,B 0,C 180,E1 -9261.589,E2 -9261.589} C_VEL
LIN {X 0,Y 432.58,Z 429.604,A -85,B 0,C 180,E1 -9264.406,E2 -9264.406} C_VEL
LIN {X 0,Y 432.604,Z 429.597,A -85,B 0,C 180,E1 -9268.138,E2 -9268.138} C_VEL
LIN {X 0,Y 432.727,Z 429.58,A -85,B 0,C 180,E1 -9270,E2 -9270} C_VEL
LIN {X 0,Y 432.58,Z 429.6,A -85,B 0,C 180,E1 -9272.793,E2 -9272.793} C_VEL
LIN {X 0,Y 432.596,Z 429.594,A -85,B 0,C 180,E1 -9275.594,E2 -9275.594} C_VEL
LIN {X 0,Y 432.465,Z 429.617,A -85,B 0,C 180,E1 -9278.41,E2 -9278.41} C_VEL
LIN {X 0,Y 432.46,Z 429.615,A -85,B 0,C 180,E1 -9282.196,E2 -9282.196} C_VEL
LIN {X 0,Y 432.431,Z 429.617,A -85,B 0,C 180,E1 -9286.039,E2 -9286.039} C_VEL
LIN {X 0,Y 432.387,Z 429.62,A -85,B 0,C 180,E1 -9289.485,E2 -9289.485} C_VEL
LIN {X 0,Y 432.318,Z 429.632,A -85,B 0,C 180,E1 -9292.964,E2 -9292.964} C_VEL
LIN {X 0,Y 432.339,Z 429.629,A -85,B 0,C 180,E1 -9295.002,E2 -9295.002} C_VEL
LIN {X 0,Y 432.347,Z 429.628,A -85,B 0,C 180,E1 -9298.125,E2 -9298.125} C_VEL
LIN {X 0,Y 432.321,Z 429.629,A -85,B 0,C 180,E1 -9301.346,E2 -9301.346} C_VEL
LIN {X 0,Y 432.339,Z 429.633,A -85,B 0,C 180,E1 -9304.677,E2 -9304.677} C_VEL
LIN {X 0,Y 432.329,Z 429.63,A -85,B 0,C 180,E1 -9308.15,E2 -9308.15} C_VEL
LIN {X 0,Y 432.323,Z 429.628,A -85,B 0,C 180,E1 -9311.6,E2 -9311.6} C_VEL
LIN {X 0,Y 432.333,Z 429.632,A -85,B 0,C 180,E1 -9314.347,E2 -9314.347} C_VEL
LIN {X 0,Y 432.315,Z 429.632,A -85,B 0,C 180,E1 -9317.016,E2 -9317.016} C_VEL
LIN {X 0,Y 432.331,Z 429.628,A -85,B 0,C 180,E1 -9319.821,E2 -9319.821} C_VEL
LIN {X 0,Y 432.304,Z 429.633,A -85,B 0,C 180,E1 -9323.022,E2 -9323.022} C_VEL
LIN {X 0,Y 432.358,Z 429.625,A -85,B 0,C 180,E1 -9325.996,E2 -9325.996} C_VEL
LIN {X 0,Y 432.347,Z 429.625,A -85,B 0,C 180,E1 -9329.49,E2 -9329.49} C_VEL
LIN {X 0,Y 432.384,Z 429.624,A -85,B 0,C 180,E1 -9332.928,E2 -9332.928} C_VEL
LIN {X 0,Y 432.366,Z 429.624,A -85,B 0,C 180,E1 -9336.023,E2 -9336.023} C_VEL
LIN {X 0,Y 432.349,Z 429.628,A -85,B 0,C 180,E1 -9339.046,E2 -9339.046} C_VEL
LIN {X 0,Y 432.36,Z 429.625,A -85,B 0,C 180,E1 -9342.01,E2 -9342.01} C_VEL
LIN {X 0,Y 432.395,Z 429.623,A -85,B 0,C 180,E1 -9344.926,E2 -9344.926} C_VEL
LIN {X 0,Y 432.459,Z 429.612,A -85,B 0,C 180,E1 -9347.803,E2 -9347.803} C_VEL
LIN {X 0,Y 432.482,Z 429.609,A -85,B 0,C 180,E1 -9351.59,E2 -9351.59} C_VEL
LIN {X 0,Y 432.586,Z 429.6,A -85,B 0,C 180,E1 -9354.406,E2 -9354.406} C_VEL
LIN {X 0,Y 432.604,Z 429.595,A -85,B 0,C 180,E1 -9358.138,E2 -9358.138} C_VEL
LIN {X 0,Y 432.732,Z 429.578,A -85,B 0,C 180,E1 -9360,E2 -9360} C_VEL
LIN {X 0,Y 432.602,Z 429.6,A -85,B 0,C 180,E1 -9362.794,E2 -9362.794} C_VEL
LIN {X 0,Y 432.572,Z 429.603,A -85,B 0,C 180,E1 -9366.53,E2 -9366.53} C_VEL
LIN {X 0,Y 432.441,Z 429.614,A -85,B 0,C 180,E1 -9369.353,E2 -9369.353} C_VEL
LIN {X 0,Y 432.431,Z 429.621,A -85,B 0,C 180,E1 -9372.804,E2 -9372.804} C_VEL
LIN {X 0,Y 432.412,Z 429.623,A -85,B 0,C 180,E1 -9376.479,E2 -9376.479} C_VEL
LIN {X 0,Y 432.338,Z 429.627,A -85,B 0,C 180,E1 -9379.961,E2 -9379.961} C_VEL
LIN {X 0,Y 432.318,Z 429.633,A -85,B 0,C 180,E1 -9382.964,E2 -9382.964} C_VEL
LIN {X 0,Y 432.343,Z 429.63,A -85,B 0,C 180,E1 -9385.002,E2 -9385.002} C_VEL
LIN {X 0,Y 432.38,Z 429.623,A -85,B 0,C 180,E1 -9388.124,E2 -9388.124} C_VEL
LIN {X 0,Y 432.321,Z 429.63,A -85,B 0,C 180,E1 -9391.346,E2 -9391.346} C_VEL
LIN {X 0,Y 432.34,Z 429.634,A -85,B 0,C 180,E1 -9394.677,E2 -9394.677} C_VEL
LIN {X 0,Y 432.336,Z 429.628,A -85,B 0,C 180,E1 -9398.15,E2 -9398.15} C_VEL
LIN {X 0,Y 432.332,Z 429.627,A -85,B 0,C 180,E1 -9401.602,E2 -9401.602} C_VEL
LIN {X 0,Y 432.334,Z 429.63,A -85,B 0,C 180,E1 -9404.348,E2 -9404.348} C_VEL
LIN {X 0,Y 432.325,Z 429.632,A -85,B 0,C 180,E1 -9407.015,E2 -9407.015} C_VEL
LIN {X 0,Y 432.337,Z 429.627,A -85,B 0,C 180,E1 -9409.821,E2 -9409.821} C_VEL
LIN {X 0,Y 432.305,Z 429.635,A -85,B 0,C 180,E1 -9413.022,E2 -9413.022} C_VEL
LIN {X 0,Y 432.36,Z 429.624,A -85,B 0,C 180,E1 -9415.997,E2 -9415.997} C_VEL
LIN {X 0,Y 432.348,Z 429.628,A -85,B 0,C 180,E1 -9419.49,E2 -9419.49} C_VEL
LIN {X 0,Y 432.412,Z 429.688,A -85,B 0,C 180,E1 -9420.818,E2 -9420.818} C_VEL
LIN {X 0,Y 435.555,Z 444.737,A -85,B 0,C 180,E1 -9423.658,E2 -9423.658} C_VEL
LIN {X 0,Y 435.9,Z 449.12,A -85,B 0,C 180,E1 -9424.441,E2 -9424.441} C_VEL
LIN {X 0,Y 434.602,Z 469.545,A -85,B 0,C 180,E1 -9427.915,E2 -9427.915} C_VEL
LIN {X 0,Y 433.627,Z 488.417,A -85,B 0,C 180,E1 -9431.086,E2 -9431.086} C_VEL
LIN {X 0,Y 433.474,Z 491.931,A -85,B 0,C 180,E1 -9431.674,E2 -9431.674} C_VEL
LIN {X 0,Y 436.795,Z 517.795,A -85,B 0,C 180,E1 -9432.312,E2 -9432.312} C_VEL
LIN {X 0,Y 435.717,Z 601.779,A -85,B 0,C 180,E1 -9433.875,E2 -9433.875} C_VEL
LIN {X 0,Y 435.159,Z 615.173,A -85,B 0,C 180,E1 -9434.305,E2 -9434.305} C_VEL
LIN {X 0,Y 434.633,Z 627.502,A -85,B 0,C 180,E1 -9434.886,E2 -9434.886} C_VEL
LIN {X 0,Y 433.971,Z 640.203,A -85,B 0,C 180,E1 -9435.702,E2 -9435.702} C_VEL
LIN {X 0,Y 433.319,Z 652.145,A -85,B 0,C 180,E1 -9436.691,E2 -9436.691} C_VEL
LIN {X 0,Y 432.783,Z 661.805,A -85,B 0,C 180,E1 -9437.694,E2 -9437.694} C_VEL
LIN {X 0,Y 432.276,Z 671.888,A -85,B 0,C 180,E1 -9438.987,E2 -9438.987} C_VEL
LIN {X 0,Y 431.837,Z 680.756,A -85,B 0,C 180,E1 -9440.398,E2 -9440.398} C_VEL
LIN {X 0,Y 431.59,Z 687.817,A -85,B 0,C 180,E1 -9441.809,E2 -9441.809} C_VEL
LIN {X 0,Y 431.383,Z 694.281,A -85,B 0,C 180,E1 -9443.452,E2 -9443.452} C_VEL
LIN {X 0,Y 431.375,Z 698.494,A -85,B 0,C 180,E1 -9444.859,E2 -9444.859} C_VEL
LIN {X 0,Y 431.326,Z 701.591,A -85,B 0,C 180,E1 -9446.263,E2 -9446.263} C_VEL
LIN {X 0,Y 431.377,Z 703.105,A -85,B 0,C 180,E1 -9447.199,E2 -9447.199} C_VEL
LIN {X 0,Y 431.404,Z 704.145,A -85,B 0,C 180,E1 -9448.133,E2 -9448.133} C_VEL
LIN {X 0,Y 431.319,Z 704.765,A -85,B 0,C 180,E1 -9449.067,E2 -9449.067} C_VEL
LIN {X 0,Y 431.296,Z 704.982,A -85,B 0,C 180,E1 -9450,E2 -9450} C_VEL
LIN {X 0,Y 431.32,Z 704.761,A -85,B 0,C 180,E1 -9450.934,E2 -9450.934} C_VEL
LIN {X 0,Y 431.406,Z 704.104,A -85,B 0,C 180,E1 -9451.867,E2 -9451.867} C_VEL
LIN {X 0,Y 431.39,Z 703.028,A -85,B 0,C 180,E1 -9452.802,E2 -9452.802} C_VEL
LIN {X 0,Y 431.334,Z 701.533,A -85,B 0,C 180,E1 -9453.737,E2 -9453.737} C_VEL
LIN {X 0,Y 431.379,Z 698.415,A -85,B 0,C 180,E1 -9455.141,E2 -9455.141} C_VEL
LIN {X 0,Y 431.385,Z 694.207,A -85,B 0,C 180,E1 -9456.549,E2 -9456.549} C_VEL
LIN {X 0,Y 431.588,Z 687.757,A -85,B 0,C 180,E1 -9458.192,E2 -9458.192} C_VEL
LIN {X 0,Y 431.838,Z 680.731,A -85,B 0,C 180,E1 -9459.603,E2 -9459.603} C_VEL
LIN {X 0,Y 432.283,Z 672.025,A -85,B 0,C 180,E1 -9461.013,E2 -9461.013} C_VEL
LIN {X 0,Y 432.773,Z 662.062,A -85,B 0,C 180,E1 -9462.307,E2 -9462.307} C_VEL
LIN {X 0,Y 433.403,Z 651.235,A -85,B 0,C 180,E1 -9463.444,E2 -9463.444} C_VEL
LIN {X 0,Y 434.11,Z 639.606,A -85,B 0,C 180,E1 -9464.414,E2 -9464.414} C_VEL
LIN {X 0,Y 434.706,Z 629.094,A -85,B 0,C 180,E1 -9465.112,E2 -9465.112} C_VEL
LIN {X 0,Y 435.404,Z 615.415,A -85,B 0,C 180,E1 -9465.807,E2 -9465.807} C_VEL
LIN {X 0,Y 436.033,Z 602.092,A -85,B 0,C 180,E1 -9466.264,E2 -9466.264} C_VEL
LIN {X 0,Y 436.3,Z 580.882,A -85,B 0,C 180,E1 -9466.705,E2 -9466.705} C_VEL
LIN {X 0,Y 437.309,Z 518.555,A -85,B 0,C 180,E1 -9467.895,E2 -9467.895} C_VEL
LIN {X 0,Y 434.448,Z 494.997,A -85,B 0,C 180,E1 -9468.517,E2 -9468.517} C_VEL
LIN {X 0,Y 433.509,Z 488.881,A -85,B 0,C 180,E1 -9468.701,E2 -9468.701} C_VEL
LIN {X 0,Y 434.47,Z 470.489,A -85,B 0,C 180,E1 -9471.842,E2 -9471.842} C_VEL
LIN {X 0,Y 435.889,Z 449.366,A -85,B 0,C 180,E1 -9475.542,E2 -9475.542} C_VEL
LIN {X 0,Y 435.73,Z 445.108,A -85,B 0,C 180,E1 -9476.331,E2 -9476.331} C_VEL
LIN {X 0,Y 433.641,Z 434.845,A -85,B 0,C 180,E1 -9478.407,E2 -9478.407} C_VEL
LIN {X 0,Y 432.357,Z 429.63,A -85,B 0,C 180,E1 -9479.521,E2 -9479.521} C_VEL
LIN {X 0,Y 432.327,Z 429.639,A -85,B 0,C 180,E1 -9482.443,E2 -9482.443} C_VEL
LIN {X 0,Y 432.348,Z 429.632,A -85,B 0,C 180,E1 -9485.632,E2 -9485.632} C_VEL
LIN {X 0,Y 432.354,Z 429.63,A -85,B 0,C 180,E1 -9489.343,E2 -9489.343} C_VEL
LIN {X 0,Y 432.337,Z 429.63,A -85,B 0,C 180,E1 -9491.797,E2 -9491.797} C_VEL
LIN {X 0,Y 432.337,Z 429.631,A -85,B 0,C 180,E1 -9494.348,E2 -9494.348} C_VEL
LIN {X 0,Y 432.32,Z 429.633,A -85,B 0,C 180,E1 -9497.016,E2 -9497.016} C_VEL
LIN {X 0,Y 432.335,Z 429.629,A -85,B 0,C 180,E1 -9499.821,E2 -9499.821} C_VEL
LIN {X 0,Y 432.308,Z 429.632,A -85,B 0,C 180,E1 -9503.022,E2 -9503.022} C_VEL
LIN {X 0,Y 432.363,Z 429.625,A -85,B 0,C 180,E1 -9505.997,E2 -9505.997} C_VEL
LIN {X 0,Y 432.35,Z 429.626,A -85,B 0,C 180,E1 -9509.49,E2 -9509.49} C_VEL
LIN {X 0,Y 432.331,Z 429.63,A -85,B 0,C 180,E1 -9511.873,E2 -9511.873} C_VEL
LIN {X 0,Y 432.357,Z 429.627,A -85,B 0,C 180,E1 -9515.546,E2 -9515.546} C_VEL
LIN {X 0,Y 432.325,Z 429.631,A -85,B 0,C 180,E1 -9519.045,E2 -9519.045} C_VEL
LIN {X 0,Y 432.318,Z 429.636,A -85,B 0,C 180,E1 -9522.008,E2 -9522.008} C_VEL
LIN {X 0,Y 432.329,Z 429.632,A -85,B 0,C 180,E1 -9524.924,E2 -9524.924} C_VEL
LIN {X 0,Y 432.451,Z 429.621,A -85,B 0,C 180,E1 -9527.803,E2 -9527.803} C_VEL
LIN {X 0,Y 432.449,Z 429.62,A -85,B 0,C 180,E1 -9531.589,E2 -9531.589} C_VEL
LIN {X 0,Y 432.55,Z 429.607,A -85,B 0,C 180,E1 -9534.405,E2 -9534.405} C_VEL
LIN {X 0,Y 432.381,Z 429.712,A -85,B 0,C 180,E1 -9535.338,E2 -9535.338} C_VEL
LIN {X 0,Y 433.171,Z 433.427,A -85,B 0,C 180,E1 -9536.384,E2 -9536.384} C_VEL
LIN {X 0,Y 437.427,Z 443.937,A -85,B 0,C 180,E1 -9536.842,E2 -9536.842} C_VEL
LIN {X 0,Y 438.071,Z 446.178,A -85,B 0,C 180,E1 -9536.925,E2 -9536.925} C_VEL
LIN {X 0,Y 436.453,Z 539.584,A -85,B 0,C 180,E1 -9538.762,E2 -9538.762} C_VEL
LIN {X 0,Y 436.163,Z 552.964,A -85,B 0,C 180,E1 -9539.224,E2 -9539.224} C_VEL
LIN {X 0,Y 435.841,Z 564.51,A -85,B 0,C 180,E1 -9539.798,E2 -9539.798} C_VEL
LIN {X 0,Y 435.259,Z 576.41,A -85,B 0,C 180,E1 -9540.578,E2 -9540.578} C_VEL
LIN {X 0,Y 434.632,Z 587.489,A -85,B 0,C 180,E1 -9541.506,E2 -9541.506} C_VEL
LIN {X 0,Y 434.018,Z 597.516,A -85,B 0,C 180,E1 -9542.552,E2 -9542.552} C_VEL
LIN {X 0,Y 433.486,Z 606.526,A -85,B 0,C 180,E1 -9543.718,E2 -9543.718} C_VEL
LIN {X 0,Y 432.915,Z 615.355,A -85,B 0,C 180,E1 -9545.123,E2 -9545.123} C_VEL
LIN {X 0,Y 432.521,Z 622.427,A -85,B 0,C 180,E1 -9546.531,E2 -9546.531} C_VEL
LIN {X 0,Y 432.11,Z 628.062,A -85,B 0,C 180,E1 -9547.946,E2 -9547.946} C_VEL
LIN {X 0,Y 431.849,Z 632.462,A -85,B 0,C 180,E1 -9549.366,E2 -9549.366} C_VEL
LIN {X 0,Y 431.684,Z 634.78,A -85,B 0,C 180,E1 -9550.316,E2 -9550.316} C_VEL
LIN {X 0,Y 431.592,Z 636.65,A -85,B 0,C 180,E1 -9551.268,E2 -9551.268} C_VEL
LIN {X 0,Y 431.485,Z 638.045,A -85,B 0,C 180,E1 -9552.235,E2 -9552.235} C_VEL
LIN {X 0,Y 431.368,Z 638.994,A -85,B 0,C 180,E1 -9553.185,E2 -9553.185} C_VEL
LIN {X 0,Y 431.346,Z 639.536,A -85,B 0,C 180,E1 -9554.146,E2 -9554.146} C_VEL
LIN {X 0,Y 431.341,Z 639.618,A -85,B 0,C 180,E1 -9555.111,E2 -9555.111} C_VEL
LIN {X 0,Y 431.356,Z 639.256,A -85,B 0,C 180,E1 -9556.08,E2 -9556.08} C_VEL
LIN {X 0,Y 431.356,Z 638.475,A -85,B 0,C 180,E1 -9557.054,E2 -9557.054} C_VEL
LIN {X 0,Y 431.395,Z 637.222,A -85,B 0,C 180,E1 -9558.031,E2 -9558.031} C_VEL
LIN {X 0,Y 431.545,Z 635.176,A -85,B 0,C 180,E1 -9559.165,E2 -9559.165} C_VEL
LIN {X 0,Y 431.677,Z 631.953,A -85,B 0,C 180,E1 -9560.489,E2 -9560.489} C_VEL
LIN {X 0,Y 431.895,Z 627.174,A -85,B 0,C 180,E1 -9561.979,E2 -9561.979} C_VEL
LIN {X 0,Y 432.242,Z 620.96,A -85,B 0,C 180,E1 -9563.475,E2 -9563.475} C_VEL
LIN {X 0,Y 432.695,Z 613,A -85,B 0,C 180,E1 -9564.98,E2 -9564.98} C_VEL
LIN {X 0,Y 433.139,Z 604.744,A -85,B 0,C 180,E1 -9566.241,E2 -9566.241} C_VEL
LIN {X 0,Y 433.66,Z 595.651,A -85,B 0,C 180,E1 -9567.378,E2 -9567.378} C_VEL
LIN {X 0,Y 434.185,Z 585.686,A -85,B 0,C 180,E1 -9568.391,E2 -9568.391} C_VEL
LIN {X 0,Y 434.744,Z 574.471,A -85,B 0,C 180,E1 -9569.31,E2 -9569.31} C_VEL
LIN {X 0,Y 435.25,Z 562.074,A -85,B 0,C 180,E1 -9570.104,E2 -9570.104} C_VEL
LIN {X 0,Y 435.646,Z 549.132,A -85,B 0,C 180,E1 -9570.71,E2 -9570.71} C_VEL
LIN {X 0,Y 435.961,Z 535.807,A -85,B 0,C 180,E1 -9571.135,E2 -9571.135} C_VEL
LIN {X 0,Y 437.187,Z 445.022,A -85,B 0,C 180,E1 -9572.825,E2 -9572.825} C_VEL
LIN {X 0,Y 432.388,Z 429.624,A -85,B 0,C 180,E1 -9573.328,E2 -9573.328} C_VEL
LIN {X 0,Y 432.337,Z 429.63,A -85,B 0,C 180,E1 -9575.818,E2 -9575.818} C_VEL
LIN {X 0,Y 432.302,Z 429.631,A -85,B 0,C 180,E1 -9579.348,E2 -9579.348} C_VEL
LIN {X 0,Y 432.311,Z 429.631,A -85,B 0,C 180,E1 -9581.8,E2 -9581.8} C_VEL
LIN {X 0,Y 432.334,Z 429.634,A -85,B 0,C 180,E1 -9584.347,E2 -9584.347} C_VEL
LIN {X 0,Y 432.305,Z 429.632,A -85,B 0,C 180,E1 -9587.018,E2 -9587.018} C_VEL
LIN {X 0,Y 432.29,Z 429.634,A -85,B 0,C 180,E1 -9589.828,E2 -9589.828} C_VEL
LIN {X 0,Y 432.299,Z 429.633,A -85,B 0,C 180,E1 -9593.021,E2 -9593.021} C_VEL
LIN {X 0,Y 432.361,Z 429.626,A -85,B 0,C 180,E1 -9595.996,E2 -9595.996} C_VEL
LIN {X 0,Y 432.348,Z 429.625,A -85,B 0,C 180,E1 -9599.49,E2 -9599.49} C_VEL
LIN {X 0,Y 432.337,Z 429.628,A -85,B 0,C 180,E1 -9601.873,E2 -9601.873} C_VEL
LIN {X 0,Y 432.378,Z 429.622,A -85,B 0,C 180,E1 -9605.539,E2 -9605.539} C_VEL
LIN {X 0,Y 432.352,Z 429.626,A -85,B 0,C 180,E1 -9609.046,E2 -9609.046} C_VEL
LIN {X 0,Y 432.359,Z 429.626,A -85,B 0,C 180,E1 -9612.01,E2 -9612.01} C_VEL
LIN {X 0,Y 432.39,Z 429.622,A -85,B 0,C 180,E1 -9614.926,E2 -9614.926} C_VEL
LIN {X 0,Y 432.381,Z 429.622,A -85,B 0,C 180,E1 -9616.59,E2 -9616.59} C_VEL
LIN {X 0,Y 431.759,Z 429.705,A -85,B 0,C 180,E1 -9617.368,E2 -9617.368} C_VEL
LIN {X 0,Y 428.938,Z 430.063,A -85,B 0,C 180,E1 -9618.631,E2 -9618.631} C_VEL
LIN {X 0,Y 426.522,Z 430.364,A -85,B 0,C 180,E1 -9619.65,E2 -9619.65} C_VEL
LIN {X 0,Y 425.478,Z 430.489,A -85,B 0,C 180,E1 -9620.438,E2 -9620.438} C_VEL
LIN {X 0,Y 425.391,Z 430.497,A -85,B 0,C 180,E1 -9620.705,E2 -9620.705} C_VEL
LIN {X 0,Y 425.482,Z 430.481,A -85,B 0,C 180,E1 -9623.36,E2 -9623.36} C_VEL
LIN {X 0,Y 425.361,Z 430.496,A -85,B 0,C 180,E1 -9625.261,E2 -9625.261} C_VEL
LIN {X 0,Y 425.573,Z 430.472,A -85,B 0,C 180,E1 -9628.107,E2 -9628.107} C_VEL
LIN {X 0,Y 425.696,Z 430.456,A -85,B 0,C 180,E1 -9630,E2 -9630} C_VEL
LIN {X 0,Y 425.533,Z 430.478,A -85,B 0,C 180,E1 -9632.84,E2 -9632.84} C_VEL
LIN {X 0,Y 425.551,Z 430.472,A -85,B 0,C 180,E1 -9635.686,E2 -9635.686} C_VEL
LIN {X 0,Y 425.409,Z 430.497,A -85,B 0,C 180,E1 -9638.55,E2 -9638.55} C_VEL
LIN {X 0,Y 425.413,Z 430.496,A -85,B 0,C 180,E1 -9642.401,E2 -9642.401} C_VEL
LIN {X 0,Y 425.389,Z 430.497,A -85,B 0,C 180,E1 -9646.311,E2 -9646.311} C_VEL
LIN {X 0,Y 425.329,Z 430.5,A -85,B 0,C 180,E1 -9649.635,E2 -9649.635} C_VEL
LIN {X 0,Y 425.288,Z 430.51,A -85,B 0,C 180,E1 -9652.338,E2 -9652.338} C_VEL
LIN {X 0,Y 425.32,Z 430.507,A -85,B 0,C 180,E1 -9654.657,E2 -9654.657} C_VEL
LIN {X 0,Y 425.272,Z 430.507,A -85,B 0,C 180,E1 -9657.563,E2 -9657.563} C_VEL
LIN {X 0,Y 425.29,Z 430.509,A -85,B 0,C 180,E1 -9660.761,E2 -9660.761} C_VEL
LIN {X 0,Y 425.311,Z 430.506,A -85,B 0,C 180,E1 -9664.288,E2 -9664.288} C_VEL
LIN {X 0,Y 425.275,Z 430.507,A -85,B 0,C 180,E1 -9667.694,E2 -9667.694} C_VEL
LIN {X 0,Y 425.265,Z 430.515,A -85,B 0,C 180,E1 -9670.518,E2 -9670.518} C_VEL
LIN {X 0,Y 425.254,Z 430.509,A -85,B 0,C 180,E1 -9673.35,E2 -9673.35} C_VEL
LIN {X 0,Y 425.26,Z 430.51,A -85,B 0,C 180,E1 -9676.044,E2 -9676.044} C_VEL
LIN {X 0,Y 425.275,Z 430.506,A -85,B 0,C 180,E1 -9679.48,E2 -9679.48} C_VEL
LIN {X 0,Y 425.275,Z 430.513,A -85,B 0,C 180,E1 -9682.489,E2 -9682.489} C_VEL
LIN {X 0,Y 425.306,Z 430.503,A -85,B 0,C 180,E1 -9685.817,E2 -9685.817} C_VEL
LIN {X 0,Y 425.29,Z 430.506,A -85,B 0,C 180,E1 -9689.239,E2 -9689.239} C_VEL
LIN {X 0,Y 425.344,Z 430.503,A -85,B 0,C 180,E1 -9692.442,E2 -9692.442} C_VEL
LIN {X 0,Y 425.346,Z 430.498,A -85,B 0,C 180,E1 -9695.602,E2 -9695.602} C_VEL
LIN {X 0,Y 425.293,Z 430.511,A -85,B 0,C 180,E1 -9698.682,E2 -9698.682} C_VEL
LIN {X 0,Y 425.321,Z 430.501,A -85,B 0,C 180,E1 -9701.702,E2 -9701.702} C_VEL
LIN {X 0,Y 425.348,Z 430.505,A -85,B 0,C 180,E1 -9704.671,E2 -9704.671} C_VEL
LIN {X 0,Y 425.411,Z 430.489,A -85,B 0,C 180,E1 -9707.598,E2 -9707.598} C_VEL
LIN {X 0,Y 425.436,Z 430.487,A -85,B 0,C 180,E1 -9711.45,E2 -9711.45} C_VEL
LIN {X 0,Y 425.541,Z 430.477,A -85,B 0,C 180,E1 -9714.313,E2 -9714.313} C_VEL
LIN {X 0,Y 425.574,Z 430.471,A -85,B 0,C 180,E1 -9718.107,E2 -9718.107} C_VEL
LIN {X 0,Y 425.701,Z 430.454,A -85,B 0,C 180,E1 -9720,E2 -9720} C_VEL
LIN {X 0,Y 425.554,Z 430.477,A -85,B 0,C 180,E1 -9722.84,E2 -9722.84} C_VEL
LIN {X 0,Y 425.531,Z 430.482,A -85,B 0,C 180,E1 -9726.639,E2 -9726.639} C_VEL
LIN {X 0,Y 425.4,Z 430.491,A -85,B 0,C 180,E1 -9729.509,E2 -9729.509} C_VEL
LIN {X 0,Y 425.393,Z 430.496,A -85,B 0,C 180,E1 -9732.904,E2 -9732.904} C_VEL
LIN {X 0,Y 425.361,Z 430.503,A -85,B 0,C 180,E1 -9736.605,E2 -9736.605} C_VEL
LIN {X 0,Y 425.328,Z 430.5,A -85,B 0,C 180,E1 -9739.636,E2 -9739.636} C_VEL
LIN {X 0,Y 425.288,Z 430.508,A -85,B 0,C 180,E1 -9742.339,E2 -9742.339} C_VEL
LIN {X 0,Y 425.322,Z 430.508,A -85,B 0,C 180,E1 -9744.658,E2 -9744.658} C_VEL
LIN {X 0,Y 425.345,Z 430.498,A -85,B 0,C 180,E1 -9747.558,E2 -9747.558} C_VEL
LIN {X 0,Y 425.287,Z 430.511,A -85,B 0,C 180,E1 -9750.816,E2 -9750.816} C_VEL
LIN {X 0,Y 425.311,Z 430.505,A -85,B 0,C 180,E1 -9754.288,E2 -9754.288} C_VEL
LIN {X 0,Y 425.278,Z 430.506,A -85,B 0,C 180,E1 -9757.695,E2 -9757.695} C_VEL
LIN {X 0,Y 425.28,Z 430.511,A -85,B 0,C 180,E1 -9760.521,E2 -9760.521} C_VEL
LIN {X 0,Y 425.257,Z 430.51,A -85,B 0,C 180,E1 -9763.351,E2 -9763.351} C_VEL
LIN {X 0,Y 425.264,Z 430.514,A -85,B 0,C 180,E1 -9766.648,E2 -9766.648} C_VEL
LIN {X 0,Y 425.29,Z 430.505,A -85,B 0,C 180,E1 -9769.873,E2 -9769.873} C_VEL
LIN {X 0,Y 425.278,Z 430.51,A -85,B 0,C 180,E1 -9772.489,E2 -9772.489} C_VEL
LIN {X 0,Y 425.308,Z 430.502,A -85,B 0,C 180,E1 -9775.818,E2 -9775.818} C_VEL
LIN {X 0,Y 425.291,Z 430.508,A -85,B 0,C 180,E1 -9779.239,E2 -9779.239} C_VEL
LIN {X 0,Y 425.377,Z 430.706,A -85,B 0,C 180,E1 -9780.606,E2 -9780.606} C_VEL
LIN {X 0,Y 428.492,Z 445.512,A -85,B 0,C 180,E1 -9783.452,E2 -9783.452} C_VEL
LIN {X 0,Y 428.977,Z 450.141,A -85,B 0,C 180,E1 -9784.3,E2 -9784.3} C_VEL
LIN {X 0,Y 427.612,Z 470.349,A -85,B 0,C 180,E1 -9787.79,E2 -9787.79} C_VEL
LIN {X 0,Y 426.67,Z 487.756,A -85,B 0,C 180,E1 -9790.766,E2 -9790.766} C_VEL
LIN {X 0,Y 426.492,Z 491.553,A -85,B 0,C 180,E1 -9791.413,E2 -9791.413} C_VEL
LIN {X 0,Y 429.949,Z 519.194,A -85,B 0,C 180,E1 -9792.091,E2 -9792.091} C_VEL
LIN {X 0,Y 428.791,Z 601.586,A -85,B 0,C 180,E1 -9793.669,E2 -9793.669} C_VEL
LIN {X 0,Y 428.202,Z 615.597,A -85,B 0,C 180,E1 -9794.135,E2 -9794.135} C_VEL
LIN {X 0,Y 427.627,Z 628.131,A -85,B 0,C 180,E1 -9794.755,E2 -9794.755} C_VEL
LIN {X 0,Y 426.947,Z 640.593,A -85,B 0,C 180,E1 -9795.584,E2 -9795.584} C_VEL
LIN {X 0,Y 426.299,Z 652.218,A -85,B 0,C 180,E1 -9796.577,E2 -9796.577} C_VEL
LIN {X 0,Y 425.734,Z 661.878,A -85,B 0,C 180,E1 -9797.608,E2 -9797.608} C_VEL
LIN {X 0,Y 425.235,Z 671.046,A -85,B 0,C 180,E1 -9798.803,E2 -9798.803} C_VEL
LIN {X 0,Y 424.787,Z 679.995,A -85,B 0,C 180,E1 -9800.237,E2 -9800.237} C_VEL
LIN {X 0,Y 424.512,Z 687.117,A -85,B 0,C 180,E1 -9801.671,E2 -9801.671} C_VEL
LIN {X 0,Y 424.303,Z 693.623,A -85,B 0,C 180,E1 -9803.342,E2 -9803.342} C_VEL
LIN {X 0,Y 424.308,Z 697.872,A -85,B 0,C 180,E1 -9804.774,E2 -9804.774} C_VEL
LIN {X 0,Y 424.235,Z 700.993,A -85,B 0,C 180,E1 -9806.201,E2 -9806.201} C_VEL
LIN {X 0,Y 424.304,Z 702.529,A -85,B 0,C 180,E1 -9807.152,E2 -9807.152} C_VEL
LIN {X 0,Y 424.331,Z 703.581,A -85,B 0,C 180,E1 -9808.102,E2 -9808.102} C_VEL
LIN {X 0,Y 424.262,Z 704.21,A -85,B 0,C 180,E1 -9809.051,E2 -9809.051} C_VEL
LIN {X 0,Y 424.237,Z 704.433,A -85,B 0,C 180,E1 -9810,E2 -9810} C_VEL
LIN {X 0,Y 424.263,Z 704.228,A -85,B 0,C 180,E1 -9810.95,E2 -9810.95} C_VEL
LIN {X 0,Y 424.32,Z 703.574,A -85,B 0,C 180,E1 -9811.899,E2 -9811.899} C_VEL
LIN {X 0,Y 424.315,Z 702.506,A -85,B 0,C 180,E1 -9812.849,E2 -9812.849} C_VEL
LIN {X 0,Y 424.239,Z 701.012,A -85,B 0,C 180,E1 -9813.8,E2 -9813.8} C_VEL
LIN {X 0,Y 424.287,Z 697.9,A -85,B 0,C 180,E1 -9815.227,E2 -9815.227} C_VEL
LIN {X 0,Y 424.308,Z 693.696,A -85,B 0,C 180,E1 -9816.658,E2 -9816.658} C_VEL
LIN {X 0,Y 424.511,Z 687.255,A -85,B 0,C 180,E1 -9818.33,E2 -9818.33} C_VEL
LIN {X 0,Y 424.803,Z 680.225,A -85,B 0,C 180,E1 -9819.764,E2 -9819.764} C_VEL
LIN {X 0,Y 425.266,Z 671.524,A -85,B 0,C 180,E1 -9821.197,E2 -9821.197} C_VEL
LIN {X 0,Y 425.723,Z 662.59,A -85,B 0,C 180,E1 -9822.393,E2 -9822.393} C_VEL
LIN {X 0,Y 426.41,Z 651.903,A -85,B 0,C 180,E1 -9823.56,E2 -9823.56} C_VEL
LIN {X 0,Y 427.112,Z 640.858,A -85,B 0,C 180,E1 -9824.533,E2 -9824.533} C_VEL
LIN {X 0,Y 427.854,Z 628.893,A -85,B 0,C 180,E1 -9825.36,E2 -9825.36} C_VEL
LIN {X 0,Y 428.565,Z 615.343,A -85,B 0,C 180,E1 -9826.066,E2 -9826.066} C_VEL
LIN {X 0,Y 429.222,Z 602.425,A -85,B 0,C 180,E1 -9826.529,E2 -9826.529} C_VEL
LIN {X 0,Y 429.511,Z 584.878,A -85,B 0,C 180,E1 -9826.915,E2 -9826.915} C_VEL
LIN {X 0,Y 430.608,Z 518.874,A -85,B 0,C 180,E1 -9828.207,E2 -9828.207} C_VEL
LIN {X 0,Y 427.949,Z 496.603,A -85,B 0,C 180,E1 -9828.824,E2 -9828.824} C_VEL
LIN {X 0,Y 426.578,Z 488.187,A -85,B 0,C 180,E1 -9829.084,E2 -9829.084} C_VEL
LIN {X 0,Y 427.521,Z 471.665,A -85,B 0,C 180,E1 -9831.962,E2 -9831.962} C_VEL
LIN {X 0,Y 428.964,Z 451.518,A -85,B 0,C 180,E1 -9835.561,E2 -9835.561} C_VEL
LIN {X 0,Y 429.03,Z 447.822,A -85,B 0,C 180,E1 -9836.251,E2 -9836.251} C_VEL
LIN {X 0,Y 426.873,Z 436.818,A -85,B 0,C 180,E1 -9838.52,E2 -9838.52} C_VEL
LIN {X 0,Y 425.323,Z 430.508,A -85,B 0,C 180,E1 -9839.922,E2 -9839.922} C_VEL
LIN {X 0,Y 425.286,Z 430.518,A -85,B 0,C 180,E1 -9843.048,E2 -9843.048} C_VEL
LIN {X 0,Y 425.286,Z 430.512,A -85,B 0,C 180,E1 -9845.929,E2 -9845.929} C_VEL
LIN {X 0,Y 425.301,Z 430.509,A -85,B 0,C 180,E1 -9849.044,E2 -9849.044} C_VEL
LIN {X 0,Y 425.278,Z 430.512,A -85,B 0,C 180,E1 -9852.653,E2 -9852.653} C_VEL
LIN {X 0,Y 425.264,Z 430.51,A -85,B 0,C 180,E1 -9856.044,E2 -9856.044} C_VEL
LIN {X 0,Y 425.28,Z 430.508,A -85,B 0,C 180,E1 -9859.481,E2 -9859.481} C_VEL
LIN {X 0,Y 425.28,Z 430.514,A -85,B 0,C 180,E1 -9862.489,E2 -9862.489} C_VEL
LIN {X 0,Y 425.311,Z 430.502,A -85,B 0,C 180,E1 -9865.817,E2 -9865.817} C_VEL
LIN {X 0,Y 425.294,Z 430.505,A -85,B 0,C 180,E1 -9869.239,E2 -9869.239} C_VEL
LIN {X 0,Y 425.255,Z 430.515,A -85,B 0,C 180,E1 -9872.436,E2 -9872.436} C_VEL
LIN {X 0,Y 425.327,Z 430.504,A -85,B 0,C 180,E1 -9875.601,E2 -9875.601} C_VEL
LIN {X 0,Y 425.277,Z 430.511,A -85,B 0,C 180,E1 -9878.681,E2 -9878.681} C_VEL
LIN {X 0,Y 425.282,Z 430.509,A -85,B 0,C 180,E1 -9881.7,E2 -9881.7} C_VEL
LIN {X 0,Y 425.281,Z 430.511,A -85,B 0,C 180,E1 -9884.668,E2 -9884.668} C_VEL
LIN {X 0,Y 425.404,Z 430.496,A -85,B 0,C 180,E1 -9887.598,E2 -9887.598} C_VEL
LIN {X 0,Y 425.397,Z 430.498,A -85,B 0,C 180,E1 -9891.449,E2 -9891.449} C_VEL
LIN {X 0,Y 425.508,Z 430.485,A -85,B 0,C 180,E1 -9894.313,E2 -9894.313} C_VEL
LIN {X 0,Y 425.404,Z 430.573,A -85,B 0,C 180,E1 -9894.965,E2 -9894.965} C_VEL
LIN {X 0,Y 426.096,Z 434.162,A -85,B 0,C 180,E1 -9895.995,E2 -9895.995} C_VEL
LIN {X 0,Y 431.286,Z 446.877,A -85,B 0,C 180,E1 -9896.568,E2 -9896.568} C_VEL
LIN {X 0,Y 431.493,Z 450.444,A -85,B 0,C 180,E1 -9896.656,E2 -9896.656} C_VEL
LIN {X 0,Y 429.717,Z 540.268,A -85,B 0,C 180,E1 -9898.477,E2 -9898.477} C_VEL
LIN {X 0,Y 429.418,Z 553.574,A -85,B 0,C 180,E1 -9898.945,E2 -9898.945} C_VEL
LIN {X 0,Y 429.007,Z 566.193,A -85,B 0,C 180,E1 -9899.592,E2 -9899.592} C_VEL
LIN {X 0,Y 428.448,Z 577.438,A -85,B 0,C 180,E1 -9900.352,E2 -9900.352} C_VEL
LIN {X 0,Y 427.798,Z 588.443,A -85,B 0,C 180,E1 -9901.294,E2 -9901.294} C_VEL
LIN {X 0,Y 427.128,Z 598.405,A -85,B 0,C 180,E1 -9902.357,E2 -9902.357} C_VEL
LIN {X 0,Y 426.569,Z 607.371,A -85,B 0,C 180,E1 -9903.542,E2 -9903.542} C_VEL
LIN {X 0,Y 425.953,Z 616.141,A -85,B 0,C 180,E1 -9904.969,E2 -9904.969} C_VEL
LIN {X 0,Y 425.532,Z 623.149,A -85,B 0,C 180,E1 -9906.401,E2 -9906.401} C_VEL
LIN {X 0,Y 425.035,Z 629.546,A -85,B 0,C 180,E1 -9908.08,E2 -9908.08} C_VEL
LIN {X 0,Y 424.779,Z 633.737,A -85,B 0,C 180,E1 -9909.523,E2 -9909.523} C_VEL
LIN {X 0,Y 424.6,Z 635.949,A -85,B 0,C 180,E1 -9910.49,E2 -9910.49} C_VEL
LIN {X 0,Y 424.399,Z 638.767,A -85,B 0,C 180,E1 -9912.301,E2 -9912.301} C_VEL
LIN {X 0,Y 424.293,Z 639.772,A -85,B 0,C 180,E1 -9913.409,E2 -9913.409} C_VEL
LIN {X 0,Y 424.259,Z 640.151,A -85,B 0,C 180,E1 -9914.388,E2 -9914.388} C_VEL
LIN {X 0,Y 424.276,Z 639.78,A -85,B 0,C 180,E1 -9916.104,E2 -9916.104} C_VEL
LIN {X 0,Y 424.298,Z 638.688,A -85,B 0,C 180,E1 -9917.346,E2 -9917.346} C_VEL
LIN {X 0,Y 424.373,Z 637.282,A -85,B 0,C 180,E1 -9918.34,E2 -9918.34} C_VEL
LIN {X 0,Y 424.555,Z 634.277,A -85,B 0,C 180,E1 -9919.837,E2 -9919.837} C_VEL
LIN {X 0,Y 424.754,Z 630.084,A -85,B 0,C 180,E1 -9921.347,E2 -9921.347} C_VEL
LIN {X 0,Y 425.018,Z 624.551,A -85,B 0,C 180,E1 -9922.867,E2 -9922.867} C_VEL
LIN {X 0,Y 425.426,Z 617.407,A -85,B 0,C 180,E1 -9924.393,E2 -9924.393} C_VEL
LIN {X 0,Y 425.853,Z 610.005,A -85,B 0,C 180,E1 -9925.672,E2 -9925.672} C_VEL
LIN {X 0,Y 426.393,Z 601.698,A -85,B 0,C 180,E1 -9926.852,E2 -9926.852} C_VEL
LIN {X 0,Y 426.876,Z 592.04,A -85,B 0,C 180,E1 -9927.984,E2 -9927.984} C_VEL
LIN {X 0,Y 427.5,Z 581.083,A -85,B 0,C 180,E1 -9929.011,E2 -9929.011} C_VEL
LIN {X 0,Y 428.048,Z 568.914,A -85,B 0,C 180,E1 -9929.915,E2 -9929.915} C_VEL
LIN {X 0,Y 428.541,Z 556.268,A -85,B 0,C 180,E1 -9930.625,E2 -9930.625} C_VEL
LIN {X 0,Y 428.923,Z 542.387,A -85,B 0,C 180,E1 -9931.176,E2 -9931.176} C_VEL
LIN {X 0,Y 429.13,Z 529.065,A -85,B 0,C 180,E1 -9931.503,E2 -9931.503} C_VEL
LIN {X 0,Y 430.347,Z 446.019,A -85,B 0,C 180,E1 -9933.065,E2 -9933.065} C_VEL
LIN {X 0,Y 425.329,Z 430.504,A -85,B 0,C 180,E1 -9933.589,E2 -9933.589} C_VEL
LIN {X 0,Y 425.262,Z 430.514,A -85,B 0,C 180,E1 -9936.509,E2 -9936.509} C_VEL
LIN {X 0,Y 425.26,Z 430.509,A -85,B 0,C 180,E1 -9939.036,E2 -9939.036} C_VEL
LIN {X 0,Y 425.263,Z 430.512,A -85,B 0,C 180,E1 -9942.655,E2 -9942.655} C_VEL
LIN {X 0,Y 425.285,Z 430.505,A -85,B 0,C 180,E1 -9945.283,E2 -9945.283} C_VEL
LIN {X 0,Y 425.25,Z 430.515,A -85,B 0,C 180,E1 -9948.618,E2 -9948.618} C_VEL
LIN {X 0,Y 425.278,Z 430.507,A -85,B 0,C 180,E1 -9951.099,E2 -9951.099} C_VEL
LIN {X 0,Y 425.298,Z 430.508,A -85,B 0,C 180,E1 -9954.663,E2 -9954.663} C_VEL
LIN {X 0,Y 425.267,Z 430.511,A -85,B 0,C 180,E1 -9958.073,E2 -9958.073} C_VEL
LIN {X 0,Y 425.307,Z 430.502,A -85,B 0,C 180,E1 -9961.366,E2 -9961.366} C_VEL
LIN {X 0,Y 425.27,Z 430.513,A -85,B 0,C 180,E1 -9964.553,E2 -9964.553} C_VEL
LIN {X 0,Y 425.306,Z 430.508,A -85,B 0,C 180,E1 -9966.634,E2 -9966.634} C_VEL
LIN {X 0,Y 425.33,Z 430.506,A -85,B 0,C 180,E1 -9970.364,E2 -9970.364} C_VEL
LIN {X 0,Y 425.387,Z 430.493,A -85,B 0,C 180,E1 -9973.688,E2 -9973.688} C_VEL
LIN {X 0,Y 425.414,Z 430.489,A -85,B 0,C 180,E1 -9977.598,E2 -9977.598} C_VEL
LIN {X 0,Y 425.391,Z 430.497,A -85,B 0,C 180,E1 -9980.705,E2 -9980.705} C_VEL
LIN {X 0,Y 424.738,Z 430.574,A -85,B 0,C 180,E1 -9981.496,E2 -9981.496} C_VEL
LIN {X 0,Y 421.95,Z 430.924,A -85,B 0,C 180,E1 -9982.782,E2 -9982.782} C_VEL
LIN {X 0,Y 419.557,Z 431.221,A -85,B 0,C 180,E1 -9983.82,E2 -9983.82} C_VEL
LIN {X 0,Y 418.48,Z 431.359,A -85,B 0,C 180,E1 -9984.621,E2 -9984.621} C_VEL
LIN {X 0,Y 418.366,Z 431.367,A -85,B 0,C 180,E1 -9984.893,E2 -9984.893} C_VEL
LIN {X 0,Y 418.542,Z 431.348,A -85,B 0,C 180,E1 -9988.075,E2 -9988.075} C_VEL
LIN {X 0,Y 418.666,Z 431.332,A -85,B 0,C 180,E1 -9990,E2 -9990} C_VEL
LIN {X 0,Y 418.489,Z 431.355,A -85,B 0,C 180,E1 -9992.888,E2 -9992.888} C_VEL
LIN {X 0,Y 418.509,Z 431.35,A -85,B 0,C 180,E1 -9995.782,E2 -9995.782} C_VEL
LIN {X 0,Y 418.379,Z 431.371,A -85,B 0,C 180,E1 -9998.695,E2 -9998.695} C_VEL
LIN {X 0,Y 418.315,Z 431.374,A -85,B 0,C 180,E1 -10001.631,E2 -10001.631} C_VEL
LIN {X 0,Y 418.304,Z 431.381,A -85,B 0,C 180,E1 -10004.597,E2 -10004.597} C_VEL
LIN {X 0,Y 418.281,Z 431.378,A -85,B 0,C 180,E1 -10007.604,E2 -10007.604} C_VEL
LIN {X 0,Y 418.251,Z 431.387,A -85,B 0,C 180,E1 -10010.663,E2 -10010.663} C_VEL
LIN {X 0,Y 418.275,Z 431.379,A -85,B 0,C 180,E1 -10013.782,E2 -10013.782} C_VEL
LIN {X 0,Y 418.227,Z 431.386,A -85,B 0,C 180,E1 -10017.048,E2 -10017.048} C_VEL
LIN {X 0,Y 418.242,Z 431.387,A -85,B 0,C 180,E1 -10020.272,E2 -10020.272} C_VEL
LIN {X 0,Y 418.248,Z 431.382,A -85,B 0,C 180,E1 -10023.677,E2 -10023.677} C_VEL
LIN {X 0,Y 418.237,Z 431.384,A -85,B 0,C 180,E1 -10027.224,E2 -10027.224} C_VEL
LIN {X 0,Y 418.216,Z 431.39,A -85,B 0,C 180,E1 -10030.869,E2 -10030.869} C_VEL
LIN {X 0,Y 418.207,Z 431.387,A -85,B 0,C 180,E1 -10033.729,E2 -10033.729} C_VEL
LIN {X 0,Y 418.207,Z 431.393,A -85,B 0,C 180,E1 -10036.448,E2 -10036.448} C_VEL
LIN {X 0,Y 418.22,Z 431.387,A -85,B 0,C 180,E1 -10039.13,E2 -10039.13} C_VEL
LIN {X 0,Y 418.224,Z 431.387,A -85,B 0,C 180,E1 -10042.167,E2 -10042.167} C_VEL
LIN {X 0,Y 418.264,Z 431.38,A -85,B 0,C 180,E1 -10045.42,E2 -10045.42} C_VEL
LIN {X 0,Y 418.212,Z 431.394,A -85,B 0,C 180,E1 -10048.604,E2 -10048.604} C_VEL
LIN {X 0,Y 418.289,Z 431.378,A -85,B 0,C 180,E1 -10051.936,E2 -10051.936} C_VEL
LIN {X 0,Y 418.271,Z 431.38,A -85,B 0,C 180,E1 -10055.161,E2 -10055.161} C_VEL
LIN {X 0,Y 418.234,Z 431.387,A -85,B 0,C 180,E1 -10058.304,E2 -10058.304} C_VEL
LIN {X 0,Y 418.275,Z 431.379,A -85,B 0,C 180,E1 -10061.383,E2 -10061.383} C_VEL
LIN {X 0,Y 418.302,Z 431.38,A -85,B 0,C 180,E1 -10064.406,E2 -10064.406} C_VEL
LIN {X 0,Y 418.355,Z 431.369,A -85,B 0,C 180,E1 -10067.386,E2 -10067.386} C_VEL
LIN {X 0,Y 418.339,Z 431.374,A -85,B 0,C 180,E1 -10070.329,E2 -10070.329} C_VEL
LIN {X 0,Y 418.463,Z 431.356,A -85,B 0,C 180,E1 -10073.249,E2 -10073.249} C_VEL
LIN {X 0,Y 418.335,Z 431.373,A -85,B 0,C 180,E1 -10075.182,E2 -10075.182} C_VEL
LIN {X 0,Y 418.543,Z 431.346,A -85,B 0,C 180,E1 -10078.076,E2 -10078.076} C_VEL
LIN {X 0,Y 418.671,Z 431.33,A -85,B 0,C 180,E1 -10080,E2 -10080} C_VEL
LIN {X 0,Y 418.507,Z 431.354,A -85,B 0,C 180,E1 -10082.888,E2 -10082.888} C_VEL
LIN {X 0,Y 418.493,Z 431.358,A -85,B 0,C 180,E1 -10086.751,E2 -10086.751} C_VEL
LIN {X 0,Y 418.4,Z 431.37,A -85,B 0,C 180,E1 -10088.695,E2 -10088.695} C_VEL
LIN {X 0,Y 418.356,Z 431.375,A -85,B 0,C 180,E1 -10092.614,E2 -10092.614} C_VEL
LIN {X 0,Y 418.302,Z 431.375,A -85,B 0,C 180,E1 -10095.594,E2 -10095.594} C_VEL
LIN {X 0,Y 418.282,Z 431.384,A -85,B 0,C 180,E1 -10098.617,E2 -10098.617} C_VEL
LIN {X 0,Y 418.234,Z 431.384,A -85,B 0,C 180,E1 -10101.697,E2 -10101.697} C_VEL
LIN {X 0,Y 418.284,Z 431.383,A -85,B 0,C 180,E1 -10104.865,E2 -10104.865} C_VEL
LIN {X 0,Y 418.289,Z 431.378,A -85,B 0,C 180,E1 -10108.064,E2 -10108.064} C_VEL
LIN {X 0,Y 418.211,Z 431.387,A -85,B 0,C 180,E1 -10111.396,E2 -10111.396} C_VEL
LIN {X 0,Y 418.265,Z 431.386,A -85,B 0,C 180,E1 -10114.58,E2 -10114.58} C_VEL
LIN {X 0,Y 418.227,Z 431.384,A -85,B 0,C 180,E1 -10117.833,E2 -10117.833} C_VEL
LIN {X 0,Y 418.222,Z 431.39,A -85,B 0,C 180,E1 -10120.948,E2 -10120.948} C_VEL
LIN {X 0,Y 418.21,Z 431.387,A -85,B 0,C 180,E1 -10123.73,E2 -10123.73} C_VEL
LIN {X 0,Y 418.216,Z 431.39,A -85,B 0,C 180,E1 -10126.45,E2 -10126.45} C_VEL
LIN {X 0,Y 418.224,Z 431.388,A -85,B 0,C 180,E1 -10129.13,E2 -10129.13} C_VEL
LIN {X 0,Y 418.228,Z 431.386,A -85,B 0,C 180,E1 -10132.167,E2 -10132.167} C_VEL
LIN {X 0,Y 418.266,Z 431.382,A -85,B 0,C 180,E1 -10135.42,E2 -10135.42} C_VEL
LIN {X 0,Y 418.213,Z 431.391,A -85,B 0,C 180,E1 -10138.604,E2 -10138.604} C_VEL
LIN {X 0,Y 418.297,Z 431.585,A -85,B 0,C 180,E1 -10140.365,E2 -10140.365} C_VEL
LIN {X 0,Y 421.429,Z 446.274,A -85,B 0,C 180,E1 -10143.239,E2 -10143.239} C_VEL
LIN {X 0,Y 422.05,Z 450.607,A -85,B 0,C 180,E1 -10144.055,E2 -10144.055} C_VEL
LIN {X 0,Y 420.758,Z 469.661,A -85,B 0,C 180,E1 -10147.408,E2 -10147.408} C_VEL
LIN {X 0,Y 419.658,Z 488.522,A -85,B 0,C 180,E1 -10150.686,E2 -10150.686} C_VEL
LIN {X 0,Y 419.533,Z 491.146,A -85,B 0,C 180,E1 -10151.14,E2 -10151.14} C_VEL
LIN {X 0,Y 423.08,Z 520.008,A -85,B 0,C 180,E1 -10151.862,E2 -10151.862} C_VEL
